// TIA Portal project "firstPro" (V15)

(* hardware
DEVICE "S71500/ET200MP station_1"  S7-1500 station
   slot 0: "导轨_0"  Rack  6ES7 590-1***0-0AA0
   slot 1: "PLC_1"  CPU 1516-3 PN/DP  6ES7 516-3AN01-0AB0  V2.5
      slot 3: "CPU 显示_1"  6ES7591-1BA00-0AA0
*)

// ===== PLC "PLC_1"  CPU 1516-3 PN/DP =====

VAR_GLOBAL   // PLC tag table "默认变量表"
   "targetdownFlag" AT %M1.0 : Bool;
   "targetupFlag" AT %M1.1 : Bool;
   "targetstopFlag" AT %M1.2 : Bool;
   "Tag_1" AT %T1 : Timer;
END_VAR

VAR_GLOBAL   // PLC tag table "变量表_1"
   "1 层上行呼梯按钮储存值" AT %I0.0 : Bool;
   "2 层上行呼梯按钮储存值" AT %I0.1 : Bool;
   "3 层上行呼梯按钮储存值" AT %I0.2 : Bool;
   "4 层上行呼梯按钮储存值" AT %I0.3 : Bool;
   "5 层上行呼梯按钮储存值" AT %I0.4 : Bool;
   "2 层下行呼梯按钮储存值" AT %I0.5 : Bool;
   "3 层下行呼梯按钮储存值" AT %I0.6 : Bool;
   "4 层下行呼梯按钮储存值" AT %I0.7 : Bool;
   "5 层下行呼梯按钮储存值" AT %I1.0 : Bool;
   "6 层下行呼梯按钮储存值" AT %I1.1 : Bool;
   "1 号梯轿内选层按钮 1储存值" AT %I1.2 : Bool;
   "1 号梯轿内选层按钮 2储存值" AT %I1.3 : Bool;
   "1 号梯轿内选层按钮 3储存值" AT %I1.4 : Bool;
   "1 号梯轿内选层按钮 4储存值" AT %I1.5 : Bool;
   "1 号梯轿内选层按钮 5储存值" AT %I1.6 : Bool;
   "1 号梯轿内选层按钮 6储存值" AT %I1.7 : Bool;
   "1层是否登记" AT %I2.0 : Bool;
   "2层是否登记" AT %I2.1 : Bool;
   "3层是否登记" AT %I2.2 : Bool;
   "4层是否登记" AT %I2.3 : Bool;
   "5层是否登记" AT %I2.4 : Bool;
   "6层是否登记" AT %I2.5 : Bool;
   "开门按钮储存值" AT %I2.6 : Bool;
   "关门按钮储存值" AT %I2.7 : Bool;
   "上平层信号储存值1" AT %I3.0 : Bool;
   "下平层信号储存值1" AT %I3.1 : Bool;
   "上平层信号储存值2" AT %I3.2 : Bool;
   "下平层信号储存值2" AT %I3.3 : Bool;
END_VAR

DATA_BLOCK "input"   // DB1
{ S7_Optimized_Access := 'FALSE' }
VERSION : 0.1
   VAR
      "1 层上行呼梯按钮" : Bool;
      "2 层上行呼梯按钮" : Bool;
      "3 层上行呼梯按钮" : Bool;
      "4 层上行呼梯按钮" : Bool;
      "5 层上行呼梯按钮" : Bool;
      "2 层下行呼梯按钮" : Bool;
      "3 层下行呼梯按钮" : Bool;
      "4 层下行呼梯按钮" : Bool;
      "5 层下行呼梯按钮" : Bool;
      "6 层下行呼梯按钮" : Bool;
      "1 号梯轿内选层按钮 1" : Bool;
      "1 号梯轿内选层按钮 2" : Bool;
      "1 号梯轿内选层按钮 3" : Bool;
      "1 号梯轿内选层按钮 4" : Bool;
      "1 号梯轿内选层按钮 5" : Bool;
      "1 号梯轿内选层按钮 6" : Bool;
      "1 号梯轿内开门按钮" : Bool;
      "1 号梯轿内关门按钮" : Bool;
      "1 号梯光幕信号" : Bool;
      "1 号梯检修信号" : Bool;
      "1 号梯轿厢门锁信号" : Bool;
      "1 号梯 1 楼层门锁信号" : Bool;
      "1 号梯 2 楼层门锁信号" : Bool;
      "1 号梯 3 楼层门锁信号" : Bool;
      "1 号梯 4 楼层门锁信号" : Bool;
      "1 号梯 5 楼层门锁信号" : Bool;
      "1 号梯 6 楼层门锁信号" : Bool;
      "1 号梯开门到位" : Bool;
      "1 号梯关门到位" : Bool;
      "1 号梯上平层信号" : Bool;
      "1 号梯下平层信号" : Bool;
      "1 号梯上端站第 1 限位" : Bool;
      "1 号梯上端站第 2 限位" : Bool;
      "1 号梯下端站第 1 限位" : Bool;
      "1 号梯下端站第 2 限位" : Bool;
      自动运行信号 : Bool;
      "1 号梯当前载重量" : Word := 0;
   END_VAR
BEGIN
END_DATA_BLOCK

DATA_BLOCK "output"   // DB2
{ S7_Optimized_Access := 'FALSE' }
VERSION : 0.1
   VAR
      "1 层上行呼梯按钮指示灯" : Bool;
      "2 层上行呼梯按钮指示灯" : Bool;
      "3 层上行呼梯按钮指示灯" : Bool;
      "4 层上行呼梯按钮指示灯" : Bool;
      "5 层上行呼梯按钮指示灯" : Bool;
      "2 层下行呼梯按钮指示灯" : Bool;
      "3 层下行呼梯按钮指示灯" : Bool;
      "4 层下行呼梯按钮指示灯" : Bool;
      "5 层下行呼梯按钮指示灯" : Bool;
      "6 层下行呼梯按钮指示灯" : Bool;
      "1 号梯 1 层按钮指示灯" : Bool;
      "1 号梯 2 层按钮指示灯" : Bool;
      "1 号梯 3 层按钮指示灯" : Bool;
      "1 号梯 4 层按钮指示灯" : Bool;
      "1 号梯 5 层按钮指示灯" : Bool;
      "1 号梯 6 层按钮指示灯" : Bool;
      "1 号梯 LEDa" : Bool;
      "1 号梯 LEDb" : Bool;
      "1 号梯 LEDc" : Bool;
      "1 号梯 LEDd" : Bool;
      "1 号梯 LEDe" : Bool;
      "1 号梯 LEDf" : Bool;
      "1 号梯 LEDg" : Bool;
      "1 号梯上行指示" : Bool;
      "1 号梯下行指示" : Bool;
      "1 号梯故障指示" : Bool;
      "1 号梯照明指示" : Bool;
      "1 号梯风扇指示" : Bool;
      "1 号梯满载指示" : Bool;
      "1 号梯电机启动信号" : Bool;
      "1 号梯上行接触器" : Bool;
      "1 号梯下行接触器" : Bool;
      "1 号梯高速接触器" : Bool;
      "1 号梯低速接触器" : Bool;
      "1 号梯开门继电器" : Bool;
      "1 号梯关门继电器" : Bool;
      "1 号梯 1 级减速制动" : Bool;
      "1 号梯 2 级减速制动" : Bool;
      "1 号梯 3 级减速制动" : Bool;
      准备就绪信号 : Bool;
   END_VAR
BEGIN
END_DATA_BLOCK

DATA_BLOCK "StateFlag"   // DB3
{ S7_Optimized_Access := 'TRUE' }
VERSION : 0.1
   VAR
      upwardFlag : Bool;
      breakingFlag : Bool;
      downwardFlag : Bool;
      startupState : UInt;
      startupflag : Bool;
      upwardState : Bool;
      downwardState : Bool;
      折返指示 : UInt;
      "1层是否登记" : Bool;
      "2层是否登记" : Bool;
      "3层是否登记" : Bool;
      "4层是否登记" : Bool;
      "5层是否登记" : Bool;
      "6层是否登记" : Bool;
      楼层是否登记 : Byte;
      重置上下行指示 : Bool := true;
      检修状态 : UInt;
   END_VAR
BEGIN
END_DATA_BLOCK

DATA_BLOCK "liftInfo"   // DB4
{ S7_Optimized_Access := 'TRUE' }
VERSION : 0.1
   VAR
      floor : Byte := 16#0;
      tartget : Byte := 16#0;
      楼层登记 : Byte;
      等待上行到达目标 : Bool;
      等待下行到达目标 : Bool;
      上行登记 : Byte;
      下行登记 : Byte;
      停层信号 : Bool;
      开门按钮储存位 : Bool;
      关门按钮储存位 : Bool;
      开门锁上下行 : Bool;
      空闲状态 : Bool := true;
      门锁信号 : Bool;
      复位空闲状态 : Bool;
      梯内按钮输入 : Byte;
      上行按钮输入 : Byte;
      下行按钮输入 : Byte;
      上下行指示 : Byte;
      上行登记掩码 : Byte := 16#3F;
      下行登记掩码 : Byte;
      检修信号 : Bool;
   END_VAR
BEGIN
END_DATA_BLOCK

DATA_BLOCK "指示灯_DB"   // DB5
{ S7_Optimized_Access := 'TRUE' }
VERSION : 0.1
// stored: InstanceOfName 指示灯
"指示灯"
BEGIN
END_DATA_BLOCK

DATA_BLOCK "constant"   // DB6
{ S7_Optimized_Access := 'TRUE' }
VERSION : 0.1
   VAR
      "1楼登记" : Byte := 16#1;
      "2楼登记" : Byte := 16#2;
      "3楼登记" : Byte := 16#4;
      "4楼登记" : Byte := 16#8;
      "5楼登记" : Byte := 16#10;
      "6楼登记" : Byte := 16#20;
      上行 : Bool := true;
      下行 : Bool;
      梯内按钮输入掩码 : Byte := 16#3F;
      上行按钮输入掩码 : Byte := 16#1F;
      下行按钮输入掩码 : Byte := 16#3F;
      楼层掩码 : Byte := 16#3F;
      上下行指示掩码 : Byte := 16#3;
      梯内按钮输入 : UInt;
      上行按钮输入 : UInt := 1;
      下行按钮输入 : UInt := 2;
      当前楼层 : UInt := 3;
      目标楼层 : UInt := 4;
      上下行指示 : UInt := 5;
      "1楼" : Byte := 16#1;
      "2楼" : Byte := 16#2;
      "3楼" : Byte := 16#4;
      "4楼" : Byte := 16#8;
      "5楼" : Byte := 16#10;
      "6楼" : Byte := 16#20;
   END_VAR
BEGIN
END_DATA_BLOCK

DATA_BLOCK "错误检测_DB"   // DB7
{ S7_Optimized_Access := 'TRUE' }
VERSION : 0.1
// stored: InstanceOfName 错误检测
"错误检测"
BEGIN
END_DATA_BLOCK

DATA_BLOCK "电梯上下行控制_DB_1"   // DB8
{ S7_Optimized_Access := 'TRUE' }
VERSION : 0.1
// stored: InstanceOfName 电梯上下行控制
"电梯上下行控制"
BEGIN
END_DATA_BLOCK

DATA_BLOCK "开关门_DB"   // DB10
{ S7_Optimized_Access := 'TRUE' }
VERSION : 0.1
// stored: InstanceOfName 开关门
"开关门"
BEGIN
END_DATA_BLOCK

DATA_BLOCK "外部信号处理储存值"   // DB16
{ S7_Optimized_Access := 'TRUE' }
VERSION : 0.1
   VAR
      梯内按钮遍历层 : Byte := 16#1;
      上行按钮遍历层 : Byte := 16#1;
      下行按钮遍历层 : Byte := 16#2;
   END_VAR
BEGIN
END_DATA_BLOCK

// folder: System blocks/Program resources

DATA_BLOCK "IEC_Timer_0_DB"   // DB9
{ S7_Optimized_Access := 'TRUE' }
AUTHOR : Simatic
FAMILY : IEC
NAME : IEC_TMR
VERSION : 1.0
// stored: InstanceOfName IEC_TIMER
"IEC_TIMER"
BEGIN
END_DATA_BLOCK

DATA_BLOCK "IEC_Timer_0_DB_2"   // DB11
{ S7_Optimized_Access := 'TRUE' }
AUTHOR : Simatic
FAMILY : IEC
NAME : IEC_TMR
VERSION : 1.0
// stored: InstanceOfName IEC_TIMER
"IEC_TIMER"
BEGIN
END_DATA_BLOCK

DATA_BLOCK "IEC_Timer_0_DB_3"   // DB12
{ S7_Optimized_Access := 'TRUE' }
AUTHOR : Simatic
FAMILY : IEC
NAME : IEC_TMR
VERSION : 1.0
// stored: InstanceOfName IEC_TIMER
"IEC_TIMER"
BEGIN
END_DATA_BLOCK

DATA_BLOCK "IEC_Timer_0_DB_4"   // DB13
{ S7_Optimized_Access := 'TRUE' }
AUTHOR : Simatic
FAMILY : IEC
NAME : IEC_TMR
VERSION : 1.0
// stored: InstanceOfName IEC_TIMER
"IEC_TIMER"
BEGIN
END_DATA_BLOCK

DATA_BLOCK "IEC_Timer_0_DB_5"   // DB14
{ S7_Optimized_Access := 'TRUE' }
AUTHOR : Simatic
FAMILY : IEC
NAME : IEC_TMR
VERSION : 1.0
// stored: InstanceOfName IEC_TIMER
"IEC_TIMER"
BEGIN
END_DATA_BLOCK

DATA_BLOCK "IEC_Timer_0_DB_1"   // DB15
{ S7_Optimized_Access := 'TRUE' }
AUTHOR : Simatic
FAMILY : IEC
NAME : IEC_TMR
VERSION : 1.0
// stored: InstanceOfName IEC_TIMER
"IEC_TIMER"
BEGIN
END_DATA_BLOCK

// folder: (top level)

FUNCTION_BLOCK "指示灯"   // FB1, LAD
{ S7_Optimized_Access := 'TRUE' }
VERSION : 0.1
   VAR_TEMP
      tmp1 : Bool;
   END_VAR
   VAR_TEMP   // added for the SCL form of the ladder/FBD networks
      _w1 : Bool;
      _w2 : Bool;
   END_VAR
BEGIN

REGION Network 1: 1层上行按钮
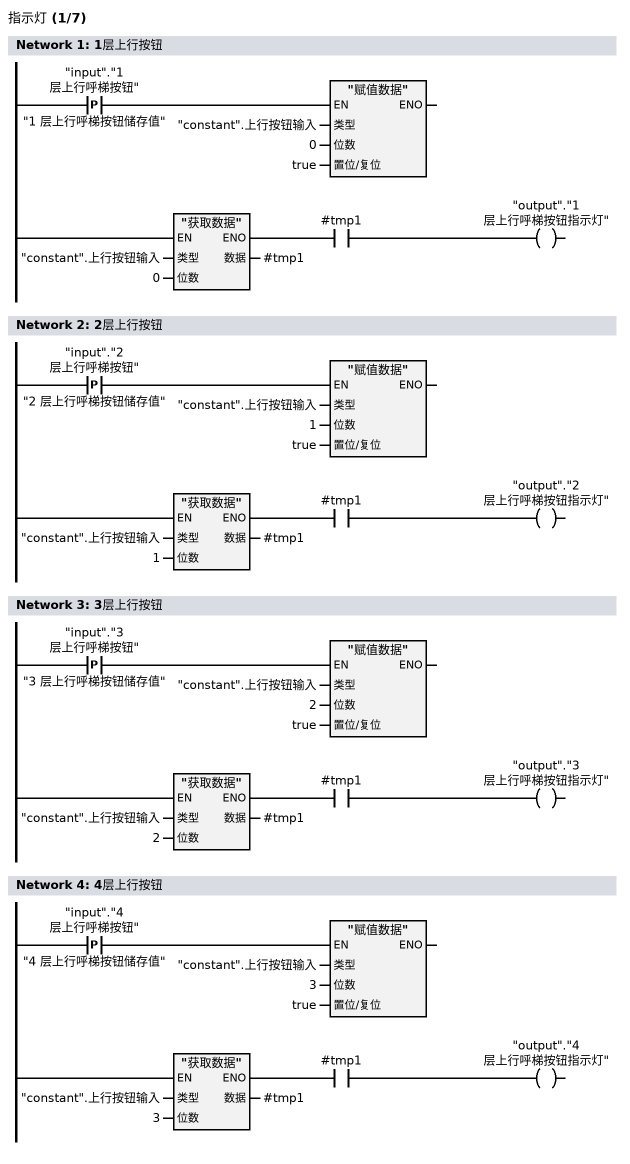
   RUNG wire#powerrail
      P_Contact(operand := "input"."1 层上行呼梯按钮", bit := "1 层上行呼梯按钮储存值")
      "赋值数据"(类型 := "constant".上行按钮输入, 位数 := 0, "置位/复位" := true)
   END_RUNG
   RUNG wire#powerrail
      "获取数据"(类型 := "constant".上行按钮输入, 位数 := 0, 数据 => #tmp1)
      Contact( #tmp1 )
      Coil( "output"."1 层上行呼梯按钮指示灯" )
   END_RUNG
   // the same network as SCL:
   #_w1 := "input"."1 层上行呼梯按钮" AND NOT "1 层上行呼梯按钮储存值";   // rising edge of "input"."1 层上行呼梯按钮"
   "1 层上行呼梯按钮储存值" := "input"."1 层上行呼梯按钮";
   IF #_w1 THEN "赋值数据"(类型 := "constant".上行按钮输入, 位数 := 0, "置位/复位" := true); END_IF;
   "获取数据"(类型 := "constant".上行按钮输入, 位数 := 0, 数据 => #tmp1, ENO => #_w2);
   "output"."1 层上行呼梯按钮指示灯" := #_w2 AND #tmp1;
END_REGION

REGION Network 2: 2层上行按钮
   RUNG wire#powerrail
      P_Contact(operand := "input"."2 层上行呼梯按钮", bit := "2 层上行呼梯按钮储存值")
      "赋值数据"(类型 := "constant".上行按钮输入, 位数 := 1, "置位/复位" := true)
   END_RUNG
   RUNG wire#powerrail
      "获取数据"(类型 := "constant".上行按钮输入, 位数 := 1, 数据 => #tmp1)
      Contact( #tmp1 )
      Coil( "output"."2 层上行呼梯按钮指示灯" )
   END_RUNG
   // the same network as SCL:
   #_w1 := "input"."2 层上行呼梯按钮" AND NOT "2 层上行呼梯按钮储存值";   // rising edge of "input"."2 层上行呼梯按钮"
   "2 层上行呼梯按钮储存值" := "input"."2 层上行呼梯按钮";
   IF #_w1 THEN "赋值数据"(类型 := "constant".上行按钮输入, 位数 := 1, "置位/复位" := true); END_IF;
   "获取数据"(类型 := "constant".上行按钮输入, 位数 := 1, 数据 => #tmp1, ENO => #_w2);
   "output"."2 层上行呼梯按钮指示灯" := #_w2 AND #tmp1;
END_REGION

REGION Network 3: 3层上行按钮
   RUNG wire#powerrail
      P_Contact(operand := "input"."3 层上行呼梯按钮", bit := "3 层上行呼梯按钮储存值")
      "赋值数据"(类型 := "constant".上行按钮输入, 位数 := 2, "置位/复位" := true)
   END_RUNG
   RUNG wire#powerrail
      "获取数据"(类型 := "constant".上行按钮输入, 位数 := 2, 数据 => #tmp1)
      Contact( #tmp1 )
      Coil( "output"."3 层上行呼梯按钮指示灯" )
   END_RUNG
   // the same network as SCL:
   #_w1 := "input"."3 层上行呼梯按钮" AND NOT "3 层上行呼梯按钮储存值";   // rising edge of "input"."3 层上行呼梯按钮"
   "3 层上行呼梯按钮储存值" := "input"."3 层上行呼梯按钮";
   IF #_w1 THEN "赋值数据"(类型 := "constant".上行按钮输入, 位数 := 2, "置位/复位" := true); END_IF;
   "获取数据"(类型 := "constant".上行按钮输入, 位数 := 2, 数据 => #tmp1, ENO => #_w2);
   "output"."3 层上行呼梯按钮指示灯" := #_w2 AND #tmp1;
END_REGION

REGION Network 4: 4层上行按钮
   RUNG wire#powerrail
      P_Contact(operand := "input"."4 层上行呼梯按钮", bit := "4 层上行呼梯按钮储存值")
      "赋值数据"(类型 := "constant".上行按钮输入, 位数 := 3, "置位/复位" := true)
   END_RUNG
   RUNG wire#powerrail
      "获取数据"(类型 := "constant".上行按钮输入, 位数 := 3, 数据 => #tmp1)
      Contact( #tmp1 )
      Coil( "output"."4 层上行呼梯按钮指示灯" )
   END_RUNG
   // the same network as SCL:
   #_w1 := "input"."4 层上行呼梯按钮" AND NOT "4 层上行呼梯按钮储存值";   // rising edge of "input"."4 层上行呼梯按钮"
   "4 层上行呼梯按钮储存值" := "input"."4 层上行呼梯按钮";
   IF #_w1 THEN "赋值数据"(类型 := "constant".上行按钮输入, 位数 := 3, "置位/复位" := true); END_IF;
   "获取数据"(类型 := "constant".上行按钮输入, 位数 := 3, 数据 => #tmp1, ENO => #_w2);
   "output"."4 层上行呼梯按钮指示灯" := #_w2 AND #tmp1;
END_REGION

REGION Network 5: 5层上行按钮
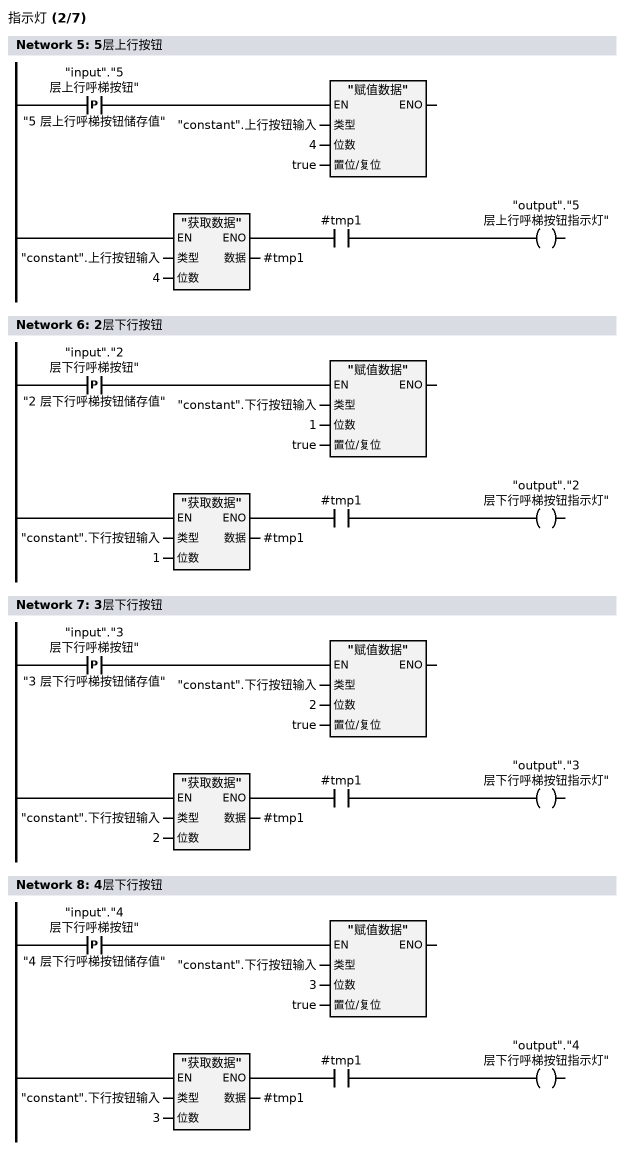
   RUNG wire#powerrail
      P_Contact(operand := "input"."5 层上行呼梯按钮", bit := "5 层上行呼梯按钮储存值")
      "赋值数据"(类型 := "constant".上行按钮输入, 位数 := 4, "置位/复位" := true)
   END_RUNG
   RUNG wire#powerrail
      "获取数据"(类型 := "constant".上行按钮输入, 位数 := 4, 数据 => #tmp1)
      Contact( #tmp1 )
      Coil( "output"."5 层上行呼梯按钮指示灯" )
   END_RUNG
   // the same network as SCL:
   #_w1 := "input"."5 层上行呼梯按钮" AND NOT "5 层上行呼梯按钮储存值";   // rising edge of "input"."5 层上行呼梯按钮"
   "5 层上行呼梯按钮储存值" := "input"."5 层上行呼梯按钮";
   IF #_w1 THEN "赋值数据"(类型 := "constant".上行按钮输入, 位数 := 4, "置位/复位" := true); END_IF;
   "获取数据"(类型 := "constant".上行按钮输入, 位数 := 4, 数据 => #tmp1, ENO => #_w2);
   "output"."5 层上行呼梯按钮指示灯" := #_w2 AND #tmp1;
END_REGION

REGION Network 6: 2层下行按钮
   RUNG wire#powerrail
      P_Contact(operand := "input"."2 层下行呼梯按钮", bit := "2 层下行呼梯按钮储存值")
      "赋值数据"(类型 := "constant".下行按钮输入, 位数 := 1, "置位/复位" := true)
   END_RUNG
   RUNG wire#powerrail
      "获取数据"(类型 := "constant".下行按钮输入, 位数 := 1, 数据 => #tmp1)
      Contact( #tmp1 )
      Coil( "output"."2 层下行呼梯按钮指示灯" )
   END_RUNG
   // the same network as SCL:
   #_w1 := "input"."2 层下行呼梯按钮" AND NOT "2 层下行呼梯按钮储存值";   // rising edge of "input"."2 层下行呼梯按钮"
   "2 层下行呼梯按钮储存值" := "input"."2 层下行呼梯按钮";
   IF #_w1 THEN "赋值数据"(类型 := "constant".下行按钮输入, 位数 := 1, "置位/复位" := true); END_IF;
   "获取数据"(类型 := "constant".下行按钮输入, 位数 := 1, 数据 => #tmp1, ENO => #_w2);
   "output"."2 层下行呼梯按钮指示灯" := #_w2 AND #tmp1;
END_REGION

REGION Network 7: 3层下行按钮
   RUNG wire#powerrail
      P_Contact(operand := "input"."3 层下行呼梯按钮", bit := "3 层下行呼梯按钮储存值")
      "赋值数据"(类型 := "constant".下行按钮输入, 位数 := 2, "置位/复位" := true)
   END_RUNG
   RUNG wire#powerrail
      "获取数据"(类型 := "constant".下行按钮输入, 位数 := 2, 数据 => #tmp1)
      Contact( #tmp1 )
      Coil( "output"."3 层下行呼梯按钮指示灯" )
   END_RUNG
   // the same network as SCL:
   #_w1 := "input"."3 层下行呼梯按钮" AND NOT "3 层下行呼梯按钮储存值";   // rising edge of "input"."3 层下行呼梯按钮"
   "3 层下行呼梯按钮储存值" := "input"."3 层下行呼梯按钮";
   IF #_w1 THEN "赋值数据"(类型 := "constant".下行按钮输入, 位数 := 2, "置位/复位" := true); END_IF;
   "获取数据"(类型 := "constant".下行按钮输入, 位数 := 2, 数据 => #tmp1, ENO => #_w2);
   "output"."3 层下行呼梯按钮指示灯" := #_w2 AND #tmp1;
END_REGION

REGION Network 8: 4层下行按钮
   RUNG wire#powerrail
      P_Contact(operand := "input"."4 层下行呼梯按钮", bit := "4 层下行呼梯按钮储存值")
      "赋值数据"(类型 := "constant".下行按钮输入, 位数 := 3, "置位/复位" := true)
   END_RUNG
   RUNG wire#powerrail
      "获取数据"(类型 := "constant".下行按钮输入, 位数 := 3, 数据 => #tmp1)
      Contact( #tmp1 )
      Coil( "output"."4 层下行呼梯按钮指示灯" )
   END_RUNG
   // the same network as SCL:
   #_w1 := "input"."4 层下行呼梯按钮" AND NOT "4 层下行呼梯按钮储存值";   // rising edge of "input"."4 层下行呼梯按钮"
   "4 层下行呼梯按钮储存值" := "input"."4 层下行呼梯按钮";
   IF #_w1 THEN "赋值数据"(类型 := "constant".下行按钮输入, 位数 := 3, "置位/复位" := true); END_IF;
   "获取数据"(类型 := "constant".下行按钮输入, 位数 := 3, 数据 => #tmp1, ENO => #_w2);
   "output"."4 层下行呼梯按钮指示灯" := #_w2 AND #tmp1;
END_REGION

REGION Network 9: 5层下行按钮
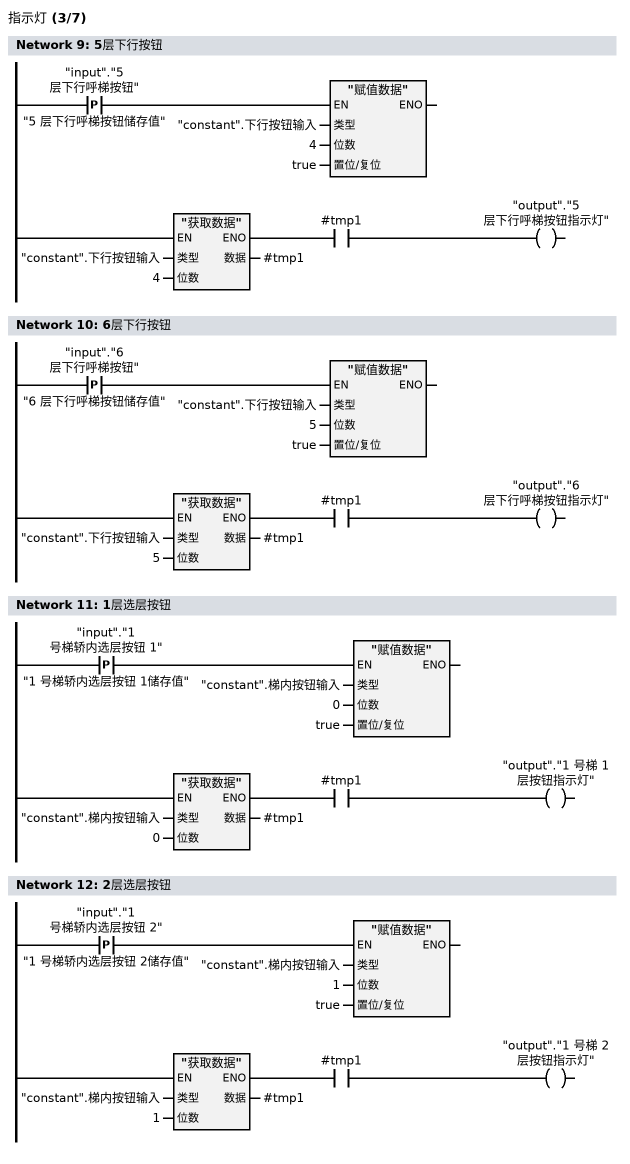
   RUNG wire#powerrail
      P_Contact(operand := "input"."5 层下行呼梯按钮", bit := "5 层下行呼梯按钮储存值")
      "赋值数据"(类型 := "constant".下行按钮输入, 位数 := 4, "置位/复位" := true)
   END_RUNG
   RUNG wire#powerrail
      "获取数据"(类型 := "constant".下行按钮输入, 位数 := 4, 数据 => #tmp1)
      Contact( #tmp1 )
      Coil( "output"."5 层下行呼梯按钮指示灯" )
   END_RUNG
   // the same network as SCL:
   #_w1 := "input"."5 层下行呼梯按钮" AND NOT "5 层下行呼梯按钮储存值";   // rising edge of "input"."5 层下行呼梯按钮"
   "5 层下行呼梯按钮储存值" := "input"."5 层下行呼梯按钮";
   IF #_w1 THEN "赋值数据"(类型 := "constant".下行按钮输入, 位数 := 4, "置位/复位" := true); END_IF;
   "获取数据"(类型 := "constant".下行按钮输入, 位数 := 4, 数据 => #tmp1, ENO => #_w2);
   "output"."5 层下行呼梯按钮指示灯" := #_w2 AND #tmp1;
END_REGION

REGION Network 10: 6层下行按钮
   RUNG wire#powerrail
      P_Contact(operand := "input"."6 层下行呼梯按钮", bit := "6 层下行呼梯按钮储存值")
      "赋值数据"(类型 := "constant".下行按钮输入, 位数 := 5, "置位/复位" := true)
   END_RUNG
   RUNG wire#powerrail
      "获取数据"(类型 := "constant".下行按钮输入, 位数 := 5, 数据 => #tmp1)
      Contact( #tmp1 )
      Coil( "output"."6 层下行呼梯按钮指示灯" )
   END_RUNG
   // the same network as SCL:
   #_w1 := "input"."6 层下行呼梯按钮" AND NOT "6 层下行呼梯按钮储存值";   // rising edge of "input"."6 层下行呼梯按钮"
   "6 层下行呼梯按钮储存值" := "input"."6 层下行呼梯按钮";
   IF #_w1 THEN "赋值数据"(类型 := "constant".下行按钮输入, 位数 := 5, "置位/复位" := true); END_IF;
   "获取数据"(类型 := "constant".下行按钮输入, 位数 := 5, 数据 => #tmp1, ENO => #_w2);
   "output"."6 层下行呼梯按钮指示灯" := #_w2 AND #tmp1;
END_REGION

REGION Network 11: 1层选层按钮
   RUNG wire#powerrail
      P_Contact(operand := "input"."1 号梯轿内选层按钮 1", bit := "1 号梯轿内选层按钮 1储存值")
      "赋值数据"(类型 := "constant".梯内按钮输入, 位数 := 0, "置位/复位" := true)
   END_RUNG
   RUNG wire#powerrail
      "获取数据"(类型 := "constant".梯内按钮输入, 位数 := 0, 数据 => #tmp1)
      Contact( #tmp1 )
      Coil( "output"."1 号梯 1 层按钮指示灯" )
   END_RUNG
   // the same network as SCL:
   #_w1 := "input"."1 号梯轿内选层按钮 1" AND NOT "1 号梯轿内选层按钮 1储存值";   // rising edge of "input"."1 号梯轿内选层按钮 1"
   "1 号梯轿内选层按钮 1储存值" := "input"."1 号梯轿内选层按钮 1";
   IF #_w1 THEN "赋值数据"(类型 := "constant".梯内按钮输入, 位数 := 0, "置位/复位" := true); END_IF;
   "获取数据"(类型 := "constant".梯内按钮输入, 位数 := 0, 数据 => #tmp1, ENO => #_w2);
   "output"."1 号梯 1 层按钮指示灯" := #_w2 AND #tmp1;
END_REGION

REGION Network 12: 2层选层按钮
   RUNG wire#powerrail
      P_Contact(operand := "input"."1 号梯轿内选层按钮 2", bit := "1 号梯轿内选层按钮 2储存值")
      "赋值数据"(类型 := "constant".梯内按钮输入, 位数 := 1, "置位/复位" := true)
   END_RUNG
   RUNG wire#powerrail
      "获取数据"(类型 := "constant".梯内按钮输入, 位数 := 1, 数据 => #tmp1)
      Contact( #tmp1 )
      Coil( "output"."1 号梯 2 层按钮指示灯" )
   END_RUNG
   // the same network as SCL:
   #_w1 := "input"."1 号梯轿内选层按钮 2" AND NOT "1 号梯轿内选层按钮 2储存值";   // rising edge of "input"."1 号梯轿内选层按钮 2"
   "1 号梯轿内选层按钮 2储存值" := "input"."1 号梯轿内选层按钮 2";
   IF #_w1 THEN "赋值数据"(类型 := "constant".梯内按钮输入, 位数 := 1, "置位/复位" := true); END_IF;
   "获取数据"(类型 := "constant".梯内按钮输入, 位数 := 1, 数据 => #tmp1, ENO => #_w2);
   "output"."1 号梯 2 层按钮指示灯" := #_w2 AND #tmp1;
END_REGION

REGION Network 13: 3层选层按钮
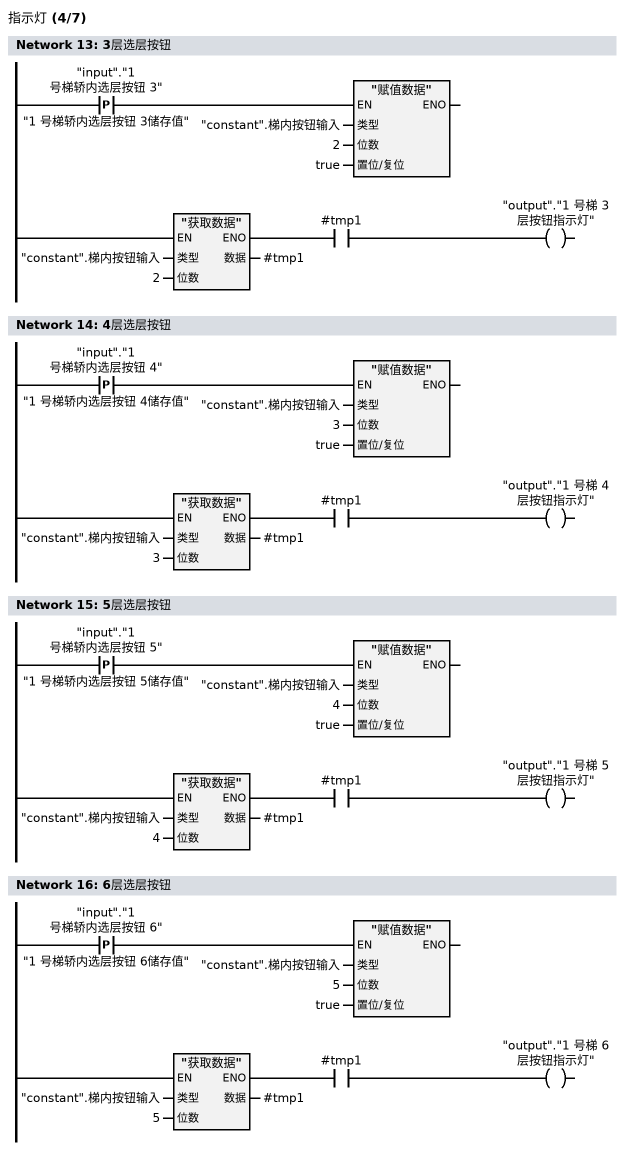
   RUNG wire#powerrail
      P_Contact(operand := "input"."1 号梯轿内选层按钮 3", bit := "1 号梯轿内选层按钮 3储存值")
      "赋值数据"(类型 := "constant".梯内按钮输入, 位数 := 2, "置位/复位" := true)
   END_RUNG
   RUNG wire#powerrail
      "获取数据"(类型 := "constant".梯内按钮输入, 位数 := 2, 数据 => #tmp1)
      Contact( #tmp1 )
      Coil( "output"."1 号梯 3 层按钮指示灯" )
   END_RUNG
   // the same network as SCL:
   #_w1 := "input"."1 号梯轿内选层按钮 3" AND NOT "1 号梯轿内选层按钮 3储存值";   // rising edge of "input"."1 号梯轿内选层按钮 3"
   "1 号梯轿内选层按钮 3储存值" := "input"."1 号梯轿内选层按钮 3";
   IF #_w1 THEN "赋值数据"(类型 := "constant".梯内按钮输入, 位数 := 2, "置位/复位" := true); END_IF;
   "获取数据"(类型 := "constant".梯内按钮输入, 位数 := 2, 数据 => #tmp1, ENO => #_w2);
   "output"."1 号梯 3 层按钮指示灯" := #_w2 AND #tmp1;
END_REGION

REGION Network 14: 4层选层按钮
   RUNG wire#powerrail
      P_Contact(operand := "input"."1 号梯轿内选层按钮 4", bit := "1 号梯轿内选层按钮 4储存值")
      "赋值数据"(类型 := "constant".梯内按钮输入, 位数 := 3, "置位/复位" := true)
   END_RUNG
   RUNG wire#powerrail
      "获取数据"(类型 := "constant".梯内按钮输入, 位数 := 3, 数据 => #tmp1)
      Contact( #tmp1 )
      Coil( "output"."1 号梯 4 层按钮指示灯" )
   END_RUNG
   // the same network as SCL:
   #_w1 := "input"."1 号梯轿内选层按钮 4" AND NOT "1 号梯轿内选层按钮 4储存值";   // rising edge of "input"."1 号梯轿内选层按钮 4"
   "1 号梯轿内选层按钮 4储存值" := "input"."1 号梯轿内选层按钮 4";
   IF #_w1 THEN "赋值数据"(类型 := "constant".梯内按钮输入, 位数 := 3, "置位/复位" := true); END_IF;
   "获取数据"(类型 := "constant".梯内按钮输入, 位数 := 3, 数据 => #tmp1, ENO => #_w2);
   "output"."1 号梯 4 层按钮指示灯" := #_w2 AND #tmp1;
END_REGION

REGION Network 15: 5层选层按钮
   RUNG wire#powerrail
      P_Contact(operand := "input"."1 号梯轿内选层按钮 5", bit := "1 号梯轿内选层按钮 5储存值")
      "赋值数据"(类型 := "constant".梯内按钮输入, 位数 := 4, "置位/复位" := true)
   END_RUNG
   RUNG wire#powerrail
      "获取数据"(类型 := "constant".梯内按钮输入, 位数 := 4, 数据 => #tmp1)
      Contact( #tmp1 )
      Coil( "output"."1 号梯 5 层按钮指示灯" )
   END_RUNG
   // the same network as SCL:
   #_w1 := "input"."1 号梯轿内选层按钮 5" AND NOT "1 号梯轿内选层按钮 5储存值";   // rising edge of "input"."1 号梯轿内选层按钮 5"
   "1 号梯轿内选层按钮 5储存值" := "input"."1 号梯轿内选层按钮 5";
   IF #_w1 THEN "赋值数据"(类型 := "constant".梯内按钮输入, 位数 := 4, "置位/复位" := true); END_IF;
   "获取数据"(类型 := "constant".梯内按钮输入, 位数 := 4, 数据 => #tmp1, ENO => #_w2);
   "output"."1 号梯 5 层按钮指示灯" := #_w2 AND #tmp1;
END_REGION

REGION Network 16: 6层选层按钮
   RUNG wire#powerrail
      P_Contact(operand := "input"."1 号梯轿内选层按钮 6", bit := "1 号梯轿内选层按钮 6储存值")
      "赋值数据"(类型 := "constant".梯内按钮输入, 位数 := 5, "置位/复位" := true)
   END_RUNG
   RUNG wire#powerrail
      "获取数据"(类型 := "constant".梯内按钮输入, 位数 := 5, 数据 => #tmp1)
      Contact( #tmp1 )
      Coil( "output"."1 号梯 6 层按钮指示灯" )
   END_RUNG
   // the same network as SCL:
   #_w1 := "input"."1 号梯轿内选层按钮 6" AND NOT "1 号梯轿内选层按钮 6储存值";   // rising edge of "input"."1 号梯轿内选层按钮 6"
   "1 号梯轿内选层按钮 6储存值" := "input"."1 号梯轿内选层按钮 6";
   IF #_w1 THEN "赋值数据"(类型 := "constant".梯内按钮输入, 位数 := 5, "置位/复位" := true); END_IF;
   "获取数据"(类型 := "constant".梯内按钮输入, 位数 := 5, 数据 => #tmp1, ENO => #_w2);
   "output"."1 号梯 6 层按钮指示灯" := #_w2 AND #tmp1;
END_REGION

REGION Network 17: One
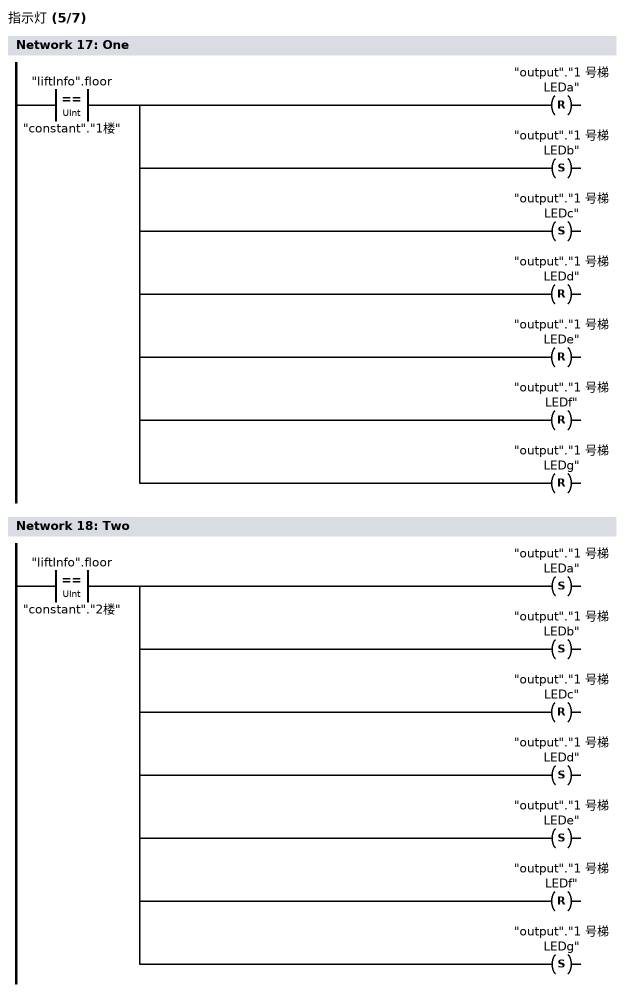
   RUNG wire#powerrail
      { S7_Templates := "SrcType := UInt" } EQ_Contact(in1 := "liftInfo".floor, in2 := "constant"."1楼")
      wire#w1
      R_Coil( "output"."1 号梯 LEDa" )
   END_RUNG
   RUNG wire#w1
      S_Coil( "output"."1 号梯 LEDb" )
   END_RUNG
   RUNG wire#w1
      S_Coil( "output"."1 号梯 LEDc" )
   END_RUNG
   RUNG wire#w1
      R_Coil( "output"."1 号梯 LEDd" )
   END_RUNG
   RUNG wire#w1
      R_Coil( "output"."1 号梯 LEDe" )
   END_RUNG
   RUNG wire#w1
      R_Coil( "output"."1 号梯 LEDf" )
   END_RUNG
   RUNG wire#w1
      R_Coil( "output"."1 号梯 LEDg" )
   END_RUNG
   // the same network as SCL:
   IF "liftInfo".floor = "constant"."1楼" THEN
       "output"."1 号梯 LEDa" := FALSE;
       "output"."1 号梯 LEDb" := TRUE;
       "output"."1 号梯 LEDc" := TRUE;
       "output"."1 号梯 LEDd" := FALSE;
       "output"."1 号梯 LEDe" := FALSE;
       "output"."1 号梯 LEDf" := FALSE;
       "output"."1 号梯 LEDg" := FALSE;
   END_IF;
END_REGION

REGION Network 18: Two
   RUNG wire#powerrail
      { S7_Templates := "SrcType := UInt" } EQ_Contact(in1 := "liftInfo".floor, in2 := "constant"."2楼")
      wire#w1
      S_Coil( "output"."1 号梯 LEDa" )
   END_RUNG
   RUNG wire#w1
      S_Coil( "output"."1 号梯 LEDb" )
   END_RUNG
   RUNG wire#w1
      R_Coil( "output"."1 号梯 LEDc" )
   END_RUNG
   RUNG wire#w1
      S_Coil( "output"."1 号梯 LEDd" )
   END_RUNG
   RUNG wire#w1
      S_Coil( "output"."1 号梯 LEDe" )
   END_RUNG
   RUNG wire#w1
      R_Coil( "output"."1 号梯 LEDf" )
   END_RUNG
   RUNG wire#w1
      S_Coil( "output"."1 号梯 LEDg" )
   END_RUNG
   // the same network as SCL:
   IF "liftInfo".floor = "constant"."2楼" THEN
       "output"."1 号梯 LEDa" := TRUE;
       "output"."1 号梯 LEDb" := TRUE;
       "output"."1 号梯 LEDc" := FALSE;
       "output"."1 号梯 LEDd" := TRUE;
       "output"."1 号梯 LEDe" := TRUE;
       "output"."1 号梯 LEDf" := FALSE;
       "output"."1 号梯 LEDg" := TRUE;
   END_IF;
END_REGION

REGION Network 19: Three
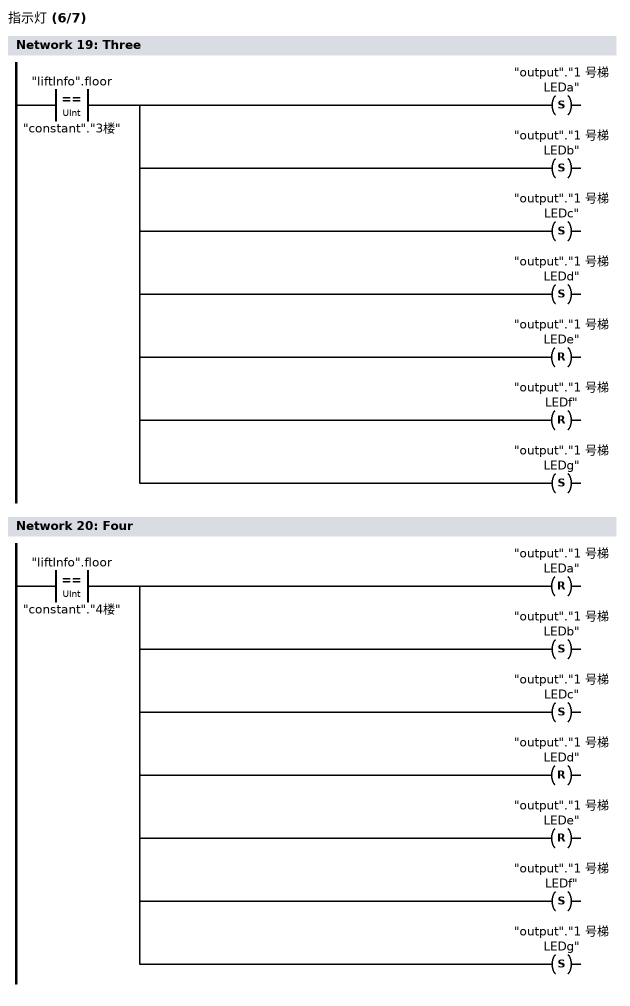
   RUNG wire#powerrail
      { S7_Templates := "SrcType := UInt" } EQ_Contact(in1 := "liftInfo".floor, in2 := "constant"."3楼")
      wire#w1
      S_Coil( "output"."1 号梯 LEDa" )
   END_RUNG
   RUNG wire#w1
      S_Coil( "output"."1 号梯 LEDb" )
   END_RUNG
   RUNG wire#w1
      S_Coil( "output"."1 号梯 LEDc" )
   END_RUNG
   RUNG wire#w1
      S_Coil( "output"."1 号梯 LEDd" )
   END_RUNG
   RUNG wire#w1
      R_Coil( "output"."1 号梯 LEDe" )
   END_RUNG
   RUNG wire#w1
      R_Coil( "output"."1 号梯 LEDf" )
   END_RUNG
   RUNG wire#w1
      S_Coil( "output"."1 号梯 LEDg" )
   END_RUNG
   // the same network as SCL:
   IF "liftInfo".floor = "constant"."3楼" THEN
       "output"."1 号梯 LEDa" := TRUE;
       "output"."1 号梯 LEDb" := TRUE;
       "output"."1 号梯 LEDc" := TRUE;
       "output"."1 号梯 LEDd" := TRUE;
       "output"."1 号梯 LEDe" := FALSE;
       "output"."1 号梯 LEDf" := FALSE;
       "output"."1 号梯 LEDg" := TRUE;
   END_IF;
END_REGION

REGION Network 20: Four
   RUNG wire#powerrail
      { S7_Templates := "SrcType := UInt" } EQ_Contact(in1 := "liftInfo".floor, in2 := "constant"."4楼")
      wire#w1
      R_Coil( "output"."1 号梯 LEDa" )
   END_RUNG
   RUNG wire#w1
      S_Coil( "output"."1 号梯 LEDb" )
   END_RUNG
   RUNG wire#w1
      S_Coil( "output"."1 号梯 LEDc" )
   END_RUNG
   RUNG wire#w1
      R_Coil( "output"."1 号梯 LEDd" )
   END_RUNG
   RUNG wire#w1
      R_Coil( "output"."1 号梯 LEDe" )
   END_RUNG
   RUNG wire#w1
      S_Coil( "output"."1 号梯 LEDf" )
   END_RUNG
   RUNG wire#w1
      S_Coil( "output"."1 号梯 LEDg" )
   END_RUNG
   // the same network as SCL:
   IF "liftInfo".floor = "constant"."4楼" THEN
       "output"."1 号梯 LEDa" := FALSE;
       "output"."1 号梯 LEDb" := TRUE;
       "output"."1 号梯 LEDc" := TRUE;
       "output"."1 号梯 LEDd" := FALSE;
       "output"."1 号梯 LEDe" := FALSE;
       "output"."1 号梯 LEDf" := TRUE;
       "output"."1 号梯 LEDg" := TRUE;
   END_IF;
END_REGION

REGION Network 21: Five
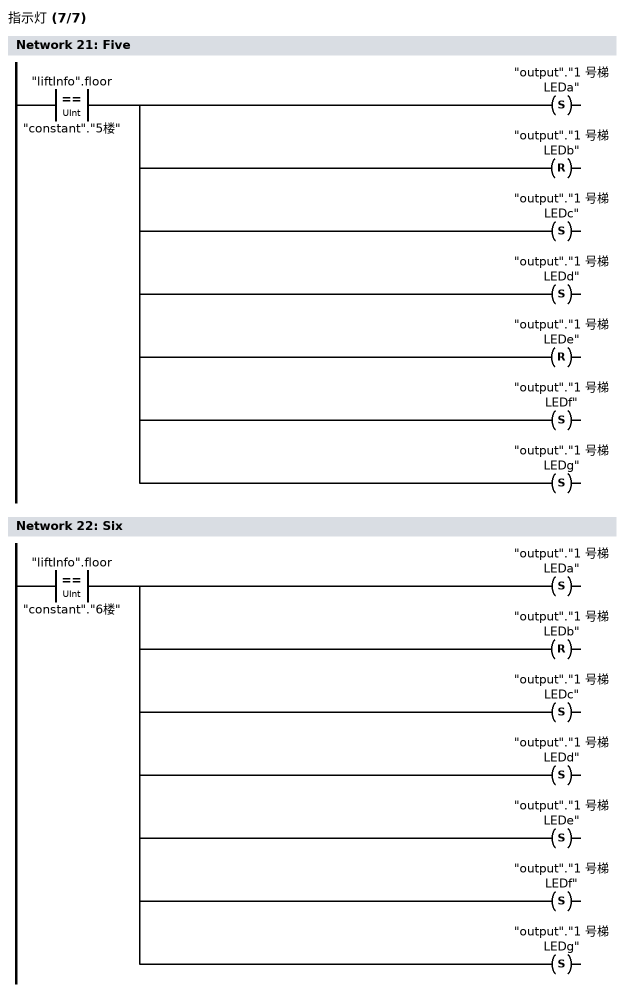
   RUNG wire#powerrail
      { S7_Templates := "SrcType := UInt" } EQ_Contact(in1 := "liftInfo".floor, in2 := "constant"."5楼")
      wire#w1
      S_Coil( "output"."1 号梯 LEDa" )
   END_RUNG
   RUNG wire#w1
      R_Coil( "output"."1 号梯 LEDb" )
   END_RUNG
   RUNG wire#w1
      S_Coil( "output"."1 号梯 LEDc" )
   END_RUNG
   RUNG wire#w1
      S_Coil( "output"."1 号梯 LEDd" )
   END_RUNG
   RUNG wire#w1
      R_Coil( "output"."1 号梯 LEDe" )
   END_RUNG
   RUNG wire#w1
      S_Coil( "output"."1 号梯 LEDf" )
   END_RUNG
   RUNG wire#w1
      S_Coil( "output"."1 号梯 LEDg" )
   END_RUNG
   // the same network as SCL:
   IF "liftInfo".floor = "constant"."5楼" THEN
       "output"."1 号梯 LEDa" := TRUE;
       "output"."1 号梯 LEDb" := FALSE;
       "output"."1 号梯 LEDc" := TRUE;
       "output"."1 号梯 LEDd" := TRUE;
       "output"."1 号梯 LEDe" := FALSE;
       "output"."1 号梯 LEDf" := TRUE;
       "output"."1 号梯 LEDg" := TRUE;
   END_IF;
END_REGION

REGION Network 22: Six
   RUNG wire#powerrail
      { S7_Templates := "SrcType := UInt" } EQ_Contact(in1 := "liftInfo".floor, in2 := "constant"."6楼")
      wire#w1
      S_Coil( "output"."1 号梯 LEDa" )
   END_RUNG
   RUNG wire#w1
      R_Coil( "output"."1 号梯 LEDb" )
   END_RUNG
   RUNG wire#w1
      S_Coil( "output"."1 号梯 LEDc" )
   END_RUNG
   RUNG wire#w1
      S_Coil( "output"."1 号梯 LEDd" )
   END_RUNG
   RUNG wire#w1
      S_Coil( "output"."1 号梯 LEDe" )
   END_RUNG
   RUNG wire#w1
      S_Coil( "output"."1 号梯 LEDf" )
   END_RUNG
   RUNG wire#w1
      S_Coil( "output"."1 号梯 LEDg" )
   END_RUNG
   // the same network as SCL:
   IF "liftInfo".floor = "constant"."6楼" THEN
       "output"."1 号梯 LEDa" := TRUE;
       "output"."1 号梯 LEDb" := FALSE;
       "output"."1 号梯 LEDc" := TRUE;
       "output"."1 号梯 LEDd" := TRUE;
       "output"."1 号梯 LEDe" := TRUE;
       "output"."1 号梯 LEDf" := TRUE;
       "output"."1 号梯 LEDg" := TRUE;
   END_IF;
END_REGION
END_FUNCTION_BLOCK

FUNCTION_BLOCK "电梯上下行控制"   // FB2, LAD
{ S7_Optimized_Access := 'TRUE' }
VERSION : 0.1
   VAR
      上行开始 : Bool;
      登记 : Byte;
      下行开始 : Bool;
      反序楼层 : UInt;
      当前楼层 : Byte;
      上升层数 : UInt;
      下行层数 : UInt;
      firstStart : Bool;
   END_VAR
   VAR_TEMP
      tmp1 : Byte;
      tmp2 : Byte;
      tmp3 : UInt;
      tmp4 : UInt;
   END_VAR
   VAR_TEMP   // added for the SCL form of the ladder/FBD networks
      _w1 : Bool;
      _w2 : Bool;
   END_VAR
BEGIN

REGION Network 1
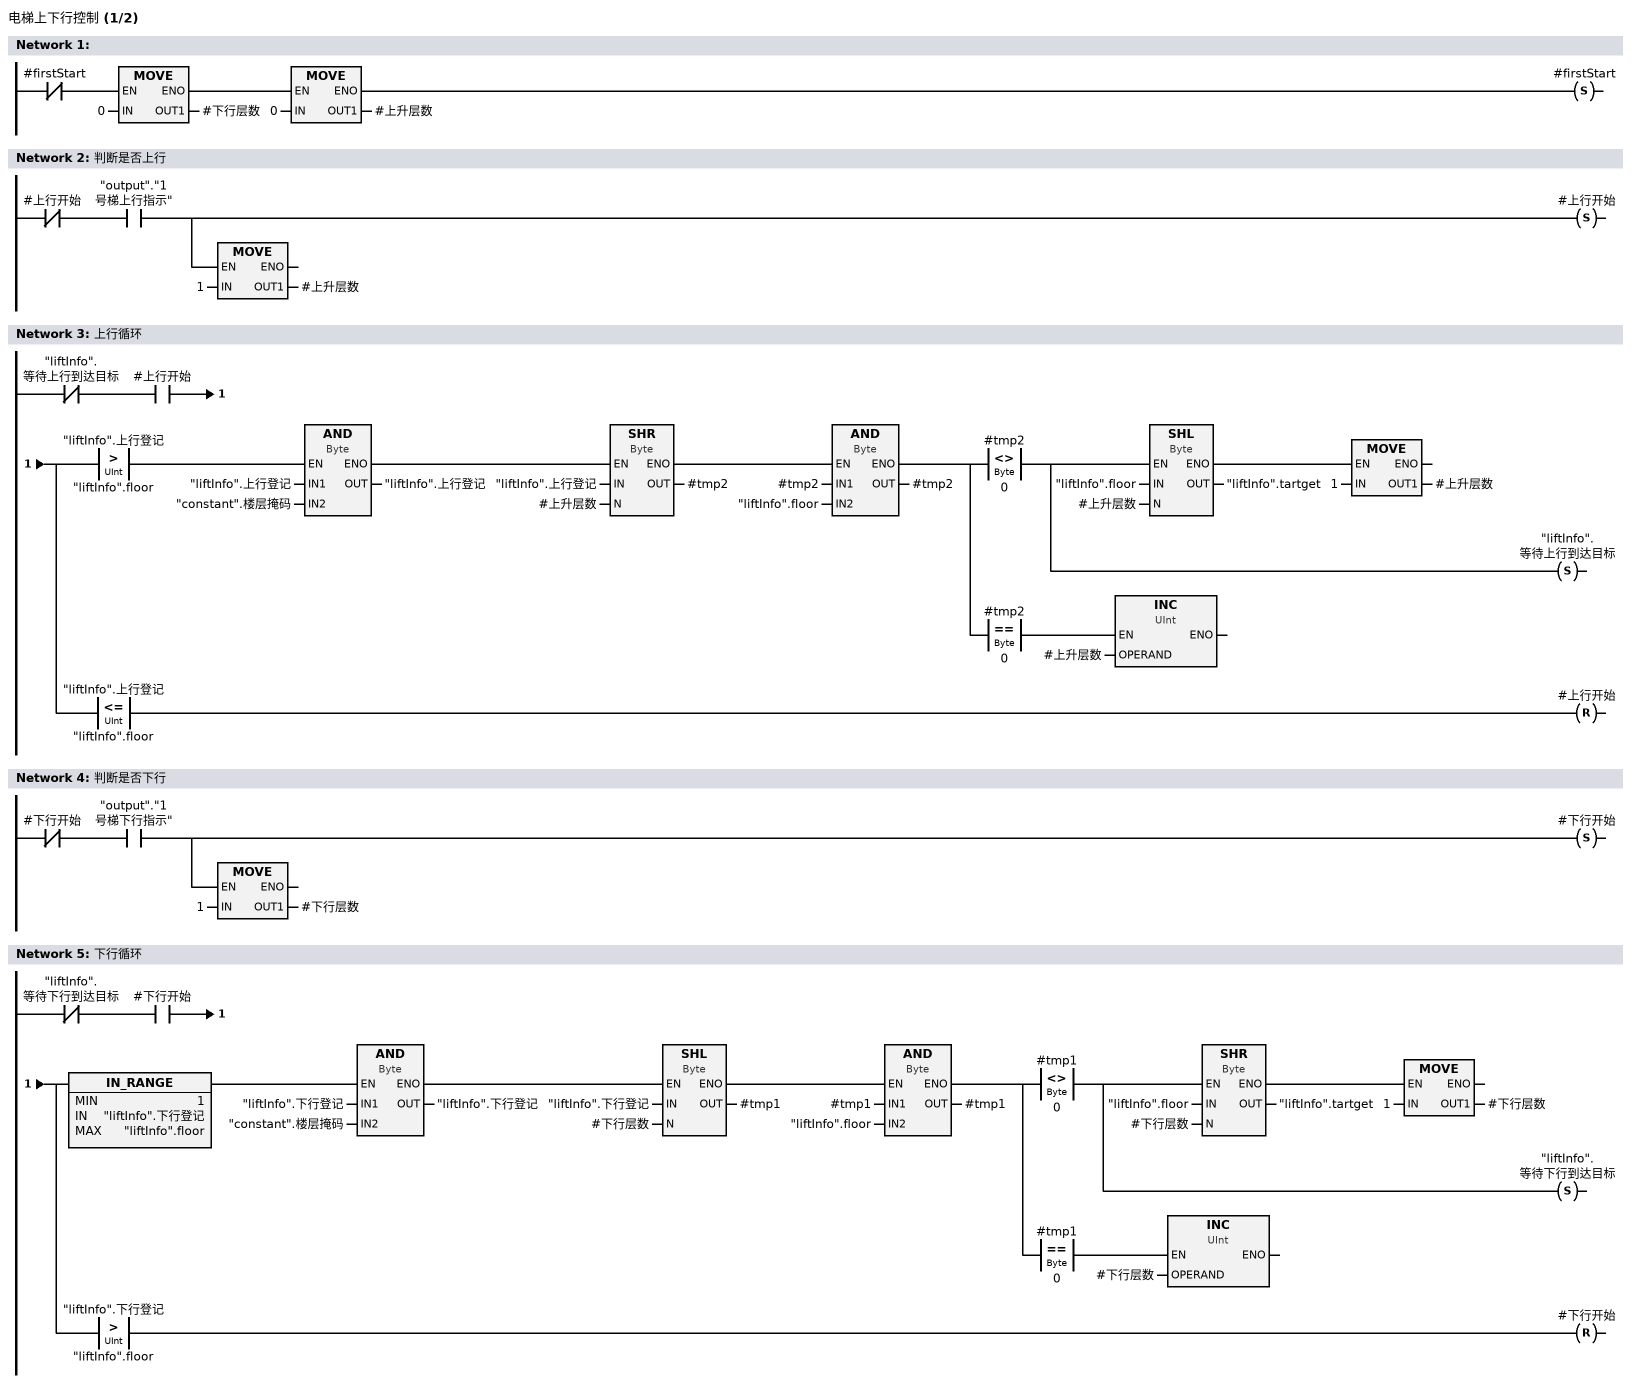
   RUNG wire#powerrail
      I_Contact( #firstStart )
      Move(in := 0, out1 => #下行层数)
      Move(in := 0, out1 => #上升层数)
      S_Coil( #firstStart )
   END_RUNG
   // the same network as SCL:
   IF NOT #firstStart THEN
       #下行层数 := 0;
       #上升层数 := 0;
       #firstStart := TRUE;
   END_IF;
END_REGION

REGION Network 2: 判断是否上行
   RUNG wire#powerrail
      I_Contact( #上行开始 )
      Contact( "output"."1 号梯上行指示" )
      wire#w1
      S_Coil( #上行开始 )
   END_RUNG
   RUNG wire#w1
      Move(in := 1, out1 => #上升层数)
   END_RUNG
   // the same network as SCL:
   #_w1 := NOT #上行开始 AND "output"."1 号梯上行指示";
   IF #_w1 THEN
       #上行开始 := TRUE;
       #上升层数 := 1;
   END_IF;
END_REGION

REGION Network 3: 上行循环
   RUNG wire#powerrail
      I_Contact( "liftInfo".等待上行到达目标 )
      Contact( #上行开始 )
      wire#w1
      { S7_Templates := "SrcType := UInt" } GT_Contact(in1 := "liftInfo".上行登记, in2 := "liftInfo".floor)
      { S7_Templates := "SrcType := Byte" } And(in1 := "liftInfo".上行登记, in2 := "constant".楼层掩码, out => "liftInfo".上行登记)
      { S7_Templates := "SrcType := Byte" } Shr(in := "liftInfo".上行登记, n := #上升层数, out => #tmp2)
      { S7_Templates := "SrcType := Byte" } And(in1 := #tmp2, in2 := "liftInfo".floor, out => #tmp2)
      wire#w2
      { S7_Templates := "SrcType := Byte" } NE_Contact(in1 := #tmp2, in2 := 0)
      wire#w3
      { S7_Templates := "SrcType := Byte" } Shl(in := "liftInfo".floor, n := #上升层数, out => "liftInfo".tartget)
      Move(in := 1, out1 => #上升层数)
   END_RUNG
   RUNG wire#w3
      S_Coil( "liftInfo".等待上行到达目标 )
   END_RUNG
   RUNG wire#w2
      { S7_Templates := "SrcType := Byte" } EQ_Contact(in1 := #tmp2, in2 := 0)
      { S7_Templates := "DestType := UInt" } Inc( #上升层数 )
   END_RUNG
   RUNG wire#w1
      { S7_Templates := "SrcType := UInt" } LE_Contact(in1 := "liftInfo".上行登记, in2 := "liftInfo".floor)
      R_Coil( #上行开始 )
   END_RUNG
   // the same network as SCL:
   #_w1 := NOT "liftInfo".等待上行到达目标 AND #上行开始;
   #_w2 := #_w1 AND ("liftInfo".上行登记 > "liftInfo".floor);
   IF #_w2 THEN
       "liftInfo".上行登记 := "liftInfo".上行登记 AND "constant".楼层掩码;
       #tmp2 := SHR(IN := "liftInfo".上行登记, N := #上升层数);
       #tmp2 := #tmp2 AND "liftInfo".floor;
   END_IF;
   IF #_w2 AND (#tmp2 <> 0) THEN
       "liftInfo".tartget := SHL(IN := "liftInfo".floor, N := #上升层数);
       #上升层数 := 1;
       "liftInfo".等待上行到达目标 := TRUE;
   END_IF;
   IF #_w2 AND (#tmp2 = 0) THEN #上升层数 := #上升层数 + 1; END_IF;
   IF #_w1 AND ("liftInfo".上行登记 <= "liftInfo".floor) THEN #上行开始 := FALSE; END_IF;
END_REGION

REGION Network 4: 判断是否下行
   RUNG wire#powerrail
      I_Contact( #下行开始 )
      Contact( "output"."1 号梯下行指示" )
      wire#w1
      S_Coil( #下行开始 )
   END_RUNG
   RUNG wire#w1
      Move(in := 1, out1 => #下行层数)
   END_RUNG
   // the same network as SCL:
   #_w1 := NOT #下行开始 AND "output"."1 号梯下行指示";
   IF #_w1 THEN
       #下行开始 := TRUE;
       #下行层数 := 1;
   END_IF;
END_REGION

REGION Network 5: 下行循环
   RUNG wire#powerrail
      I_Contact( "liftInfo".等待下行到达目标 )
      Contact( #下行开始 )
      wire#w1
      { S7_Templates := "SrcType := UInt" } InRange(min := 1, in := "liftInfo".下行登记, max := "liftInfo".floor)
      { S7_Templates := "SrcType := Byte" } And(in1 := "liftInfo".下行登记, in2 := "constant".楼层掩码, out => "liftInfo".下行登记)
      { S7_Templates := "SrcType := Byte" } Shl(in := "liftInfo".下行登记, n := #下行层数, out => #tmp1)
      { S7_Templates := "SrcType := Byte" } And(in1 := #tmp1, in2 := "liftInfo".floor, out => #tmp1)
      wire#w2
      { S7_Templates := "SrcType := Byte" } NE_Contact(in1 := #tmp1, in2 := 0)
      wire#w3
      { S7_Templates := "SrcType := Byte" } Shr(in := "liftInfo".floor, n := #下行层数, out => "liftInfo".tartget)
      Move(in := 1, out1 => #下行层数)
   END_RUNG
   RUNG wire#w3
      S_Coil( "liftInfo".等待下行到达目标 )
   END_RUNG
   RUNG wire#w2
      { S7_Templates := "SrcType := Byte" } EQ_Contact(in1 := #tmp1, in2 := 0)
      { S7_Templates := "DestType := UInt" } Inc( #下行层数 )
   END_RUNG
   RUNG wire#w1
      { S7_Templates := "SrcType := UInt" } GT_Contact(in1 := "liftInfo".下行登记, in2 := "liftInfo".floor)
      R_Coil( #下行开始 )
   END_RUNG
   // the same network as SCL:
   #_w1 := NOT "liftInfo".等待下行到达目标 AND #下行开始;
   #_w2 := #_w1 AND (1 <= "liftInfo".下行登记) AND ("liftInfo".下行登记 <= "liftInfo".floor);
   IF #_w2 THEN
       "liftInfo".下行登记 := "liftInfo".下行登记 AND "constant".楼层掩码;
       #tmp1 := SHL(IN := "liftInfo".下行登记, N := #下行层数);
       #tmp1 := #tmp1 AND "liftInfo".floor;
   END_IF;
   IF #_w2 AND (#tmp1 <> 0) THEN
       "liftInfo".tartget := SHR(IN := "liftInfo".floor, N := #下行层数);
       #下行层数 := 1;
       "liftInfo".等待下行到达目标 := TRUE;
   END_IF;
   IF #_w2 AND (#tmp1 = 0) THEN #下行层数 := #下行层数 + 1; END_IF;
   IF #_w1 AND ("liftInfo".下行登记 > "liftInfo".floor) THEN #下行开始 := FALSE; END_IF;
END_REGION

REGION Network 6: 静止时，判断上下行
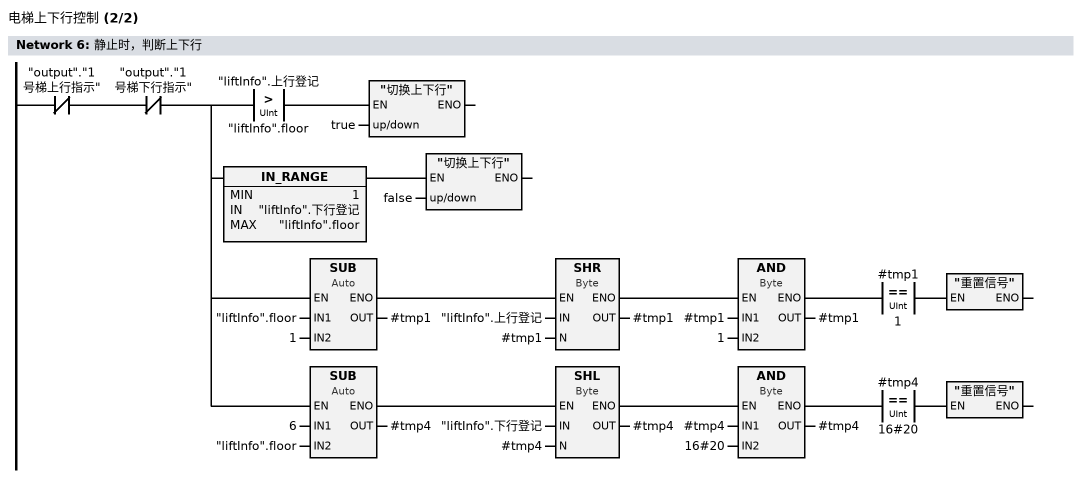
   RUNG wire#powerrail
      I_Contact( "output"."1 号梯上行指示" )
      I_Contact( "output"."1 号梯下行指示" )
      wire#w1
      { S7_Templates := "SrcType := UInt" } GT_Contact(in1 := "liftInfo".上行登记, in2 := "liftInfo".floor)
      "切换上下行"("up/down" := true)
   END_RUNG
   RUNG wire#w1
      { S7_Templates := "SrcType := UInt" } InRange(min := 1, in := "liftInfo".下行登记, max := "liftInfo".floor)
      "切换上下行"("up/down" := false)
   END_RUNG
   RUNG wire#w1
      Sub(in1 := "liftInfo".floor, in2 := 1, out => #tmp1)
      { S7_Templates := "SrcType := Byte" } Shr(in := "liftInfo".上行登记, n := #tmp1, out => #tmp1)
      { S7_Templates := "SrcType := Byte" } And(in1 := #tmp1, in2 := 1, out => #tmp1)
      { S7_Templates := "SrcType := UInt" } EQ_Contact(in1 := #tmp1, in2 := 1)
      "重置信号"()
   END_RUNG
   RUNG wire#w1
      Sub(in1 := 6, in2 := "liftInfo".floor, out => #tmp4)
      { S7_Templates := "SrcType := Byte" } Shl(in := "liftInfo".下行登记, n := #tmp4, out => #tmp4)
      { S7_Templates := "SrcType := Byte" } And(in1 := #tmp4, in2 := 16#20, out => #tmp4)
      { S7_Templates := "SrcType := UInt" } EQ_Contact(in1 := #tmp4, in2 := 16#20)
      "重置信号"()
   END_RUNG
   // the same network as SCL:
   #_w1 := NOT "output"."1 号梯上行指示" AND NOT "output"."1 号梯下行指示";
   IF #_w1 AND ("liftInfo".上行登记 > "liftInfo".floor) THEN "切换上下行"("up/down" := true); END_IF;
   IF #_w1 AND (1 <= "liftInfo".下行登记) AND ("liftInfo".下行登记 <= "liftInfo".floor) THEN
       "切换上下行"("up/down" := false);
   END_IF;
   IF #_w1 THEN
       #tmp1 := "liftInfo".floor - 1;
       #tmp1 := SHR(IN := "liftInfo".上行登记, N := #tmp1);
       #tmp1 := #tmp1 AND 1;
   END_IF;
   IF #_w1 AND (#tmp1 = 1) THEN "重置信号"(); END_IF;
   IF #_w1 THEN
       #tmp4 := 6 - "liftInfo".floor;
       #tmp4 := SHL(IN := "liftInfo".下行登记, N := #tmp4);
       #tmp4 := #tmp4 AND 16#20;
   END_IF;
   IF #_w1 AND (#tmp4 = 16#20) THEN "重置信号"(); END_IF;
END_REGION
END_FUNCTION_BLOCK

FUNCTION_BLOCK "错误检测"   // FB3, LAD
{ S7_Optimized_Access := 'TRUE' }
VERSION : 0.1
   VAR_TEMP   // added for the SCL form of the ladder/FBD networks
      _w1 : Bool;
   END_VAR
BEGIN

REGION Network 1
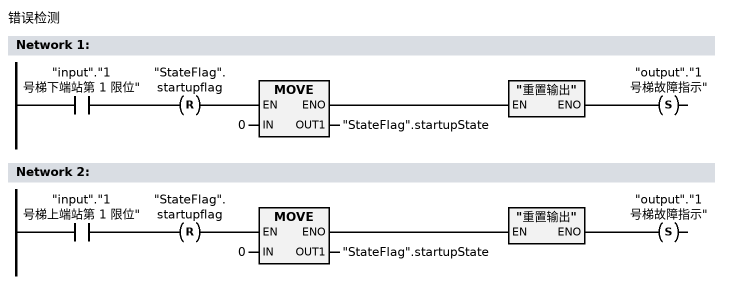
   RUNG wire#powerrail
      Contact( "input"."1 号梯下端站第 1 限位" )
      R_Coil( "StateFlag".startupflag )
      Move(in := 0, out1 => "StateFlag".startupState)
      "重置输出"()
      S_Coil( "output"."1 号梯故障指示" )
   END_RUNG
   // the same network as SCL:
   IF "input"."1 号梯下端站第 1 限位" THEN
       "StateFlag".startupflag := FALSE;
       "StateFlag".startupState := 0;
   END_IF;
   "重置输出"(EN := "input"."1 号梯下端站第 1 限位", ENO => #_w1);
   IF #_w1 THEN "output"."1 号梯故障指示" := TRUE; END_IF;
END_REGION

REGION Network 2
   RUNG wire#powerrail
      Contact( "input"."1 号梯上端站第 1 限位" )
      R_Coil( "StateFlag".startupflag )
      Move(in := 0, out1 => "StateFlag".startupState)
      "重置输出"()
      S_Coil( "output"."1 号梯故障指示" )
   END_RUNG
   // the same network as SCL:
   IF "input"."1 号梯上端站第 1 限位" THEN
       "StateFlag".startupflag := FALSE;
       "StateFlag".startupState := 0;
   END_IF;
   "重置输出"(EN := "input"."1 号梯上端站第 1 限位", ENO => #_w1);
   IF #_w1 THEN "output"."1 号梯故障指示" := TRUE; END_IF;
END_REGION
END_FUNCTION_BLOCK

FUNCTION_BLOCK "开关门"   // FB4, LAD
{ S7_Optimized_Access := 'TRUE' }
VERSION : 0.1
   VAR_TEMP   // added for the SCL form of the ladder/FBD networks
      _w1 : Bool;
      _w2 : Bool;
   END_VAR
BEGIN

REGION Network 1: 按键开门
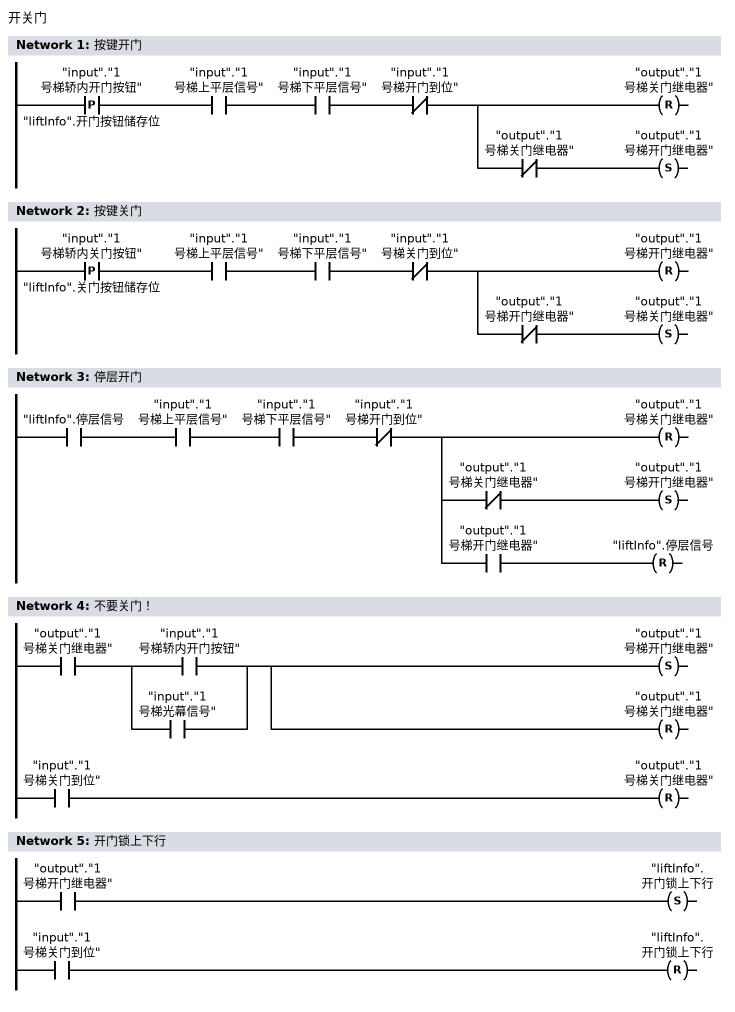
   RUNG wire#powerrail
      P_Contact(operand := "input"."1 号梯轿内开门按钮", bit := "liftInfo".开门按钮储存位)
      Contact( "input"."1 号梯上平层信号" )
      Contact( "input"."1 号梯下平层信号" )
      I_Contact( "input"."1 号梯开门到位" )
      wire#w1
      R_Coil( "output"."1 号梯关门继电器" )
   END_RUNG
   RUNG wire#w1
      I_Contact( "output"."1 号梯关门继电器" )
      S_Coil( "output"."1 号梯开门继电器" )
   END_RUNG
   // the same network as SCL:
   #_w1 := "input"."1 号梯轿内开门按钮" AND NOT "liftInfo".开门按钮储存位;   // rising edge of "input"."1 号梯轿内开门按钮"
   "liftInfo".开门按钮储存位 := "input"."1 号梯轿内开门按钮";
   #_w2 := #_w1 AND "input"."1 号梯上平层信号" AND "input"."1 号梯下平层信号" AND NOT "input"."1 号梯开门到位";
   IF #_w2 THEN "output"."1 号梯关门继电器" := FALSE; END_IF;
   IF #_w2 AND NOT "output"."1 号梯关门继电器" THEN "output"."1 号梯开门继电器" := TRUE; END_IF;
END_REGION

REGION Network 2: 按键关门
   RUNG wire#powerrail
      P_Contact(operand := "input"."1 号梯轿内关门按钮", bit := "liftInfo".关门按钮储存位)
      Contact( "input"."1 号梯上平层信号" )
      Contact( "input"."1 号梯下平层信号" )
      I_Contact( "input"."1 号梯关门到位" )
      wire#w1
      R_Coil( "output"."1 号梯开门继电器" )
   END_RUNG
   RUNG wire#w1
      I_Contact( "output"."1 号梯开门继电器" )
      S_Coil( "output"."1 号梯关门继电器" )
   END_RUNG
   // the same network as SCL:
   #_w1 := "input"."1 号梯轿内关门按钮" AND NOT "liftInfo".关门按钮储存位;   // rising edge of "input"."1 号梯轿内关门按钮"
   "liftInfo".关门按钮储存位 := "input"."1 号梯轿内关门按钮";
   #_w2 := #_w1 AND "input"."1 号梯上平层信号" AND "input"."1 号梯下平层信号" AND NOT "input"."1 号梯关门到位";
   IF #_w2 THEN "output"."1 号梯开门继电器" := FALSE; END_IF;
   IF #_w2 AND NOT "output"."1 号梯开门继电器" THEN "output"."1 号梯关门继电器" := TRUE; END_IF;
END_REGION

REGION Network 3: 停层开门
   RUNG wire#powerrail
      Contact( "liftInfo".停层信号 )
      Contact( "input"."1 号梯上平层信号" )
      Contact( "input"."1 号梯下平层信号" )
      I_Contact( "input"."1 号梯开门到位" )
      wire#w1
      R_Coil( "output"."1 号梯关门继电器" )
   END_RUNG
   RUNG wire#w1
      I_Contact( "output"."1 号梯关门继电器" )
      S_Coil( "output"."1 号梯开门继电器" )
   END_RUNG
   RUNG wire#w1
      Contact( "output"."1 号梯开门继电器" )
      R_Coil( "liftInfo".停层信号 )
   END_RUNG
   // the same network as SCL:
   #_w1 := "liftInfo".停层信号 AND "input"."1 号梯上平层信号" AND "input"."1 号梯下平层信号" AND NOT "input"."1 号梯开门到位";
   IF #_w1 THEN "output"."1 号梯关门继电器" := FALSE; END_IF;
   IF #_w1 AND NOT "output"."1 号梯关门继电器" THEN "output"."1 号梯开门继电器" := TRUE; END_IF;
   IF #_w1 AND "output"."1 号梯开门继电器" THEN "liftInfo".停层信号 := FALSE; END_IF;
END_REGION

REGION Network 4: 不要关门！
   RUNG wire#powerrail
      Contact( "output"."1 号梯关门继电器" )
      wire#w1
      Contact( "input"."1 号梯轿内开门按钮" )
      wire#w2
      S_Coil( "output"."1 号梯开门继电器" )
   END_RUNG
   RUNG wire#w1
      Contact( "input"."1 号梯光幕信号" )
   END_RUNG wire#w2
   RUNG wire#w2
      R_Coil( "output"."1 号梯关门继电器" )
   END_RUNG
   RUNG wire#powerrail
      Contact( "input"."1 号梯关门到位" )
      R_Coil( "output"."1 号梯关门继电器" )
   END_RUNG
   // the same network as SCL:
   IF "output"."1 号梯关门继电器" AND ("input"."1 号梯轿内开门按钮" OR "input"."1 号梯光幕信号") THEN
       "output"."1 号梯开门继电器" := TRUE;
       "output"."1 号梯关门继电器" := FALSE;
   END_IF;
   IF "input"."1 号梯关门到位" THEN "output"."1 号梯关门继电器" := FALSE; END_IF;
END_REGION

REGION Network 5: 开门锁上下行
   RUNG wire#powerrail
      Contact( "output"."1 号梯开门继电器" )
      S_Coil( "liftInfo".开门锁上下行 )
   END_RUNG
   RUNG wire#powerrail
      Contact( "input"."1 号梯关门到位" )
      R_Coil( "liftInfo".开门锁上下行 )
   END_RUNG
   // the same network as SCL:
   IF "output"."1 号梯开门继电器" THEN "liftInfo".开门锁上下行 := TRUE; END_IF;
   IF "input"."1 号梯关门到位" THEN "liftInfo".开门锁上下行 := FALSE; END_IF;
END_REGION
END_FUNCTION_BLOCK

FUNCTION "赋值数据" : Void   // FC1, LAD
{ S7_Optimized_Access := 'TRUE' }
VERSION : 0.1
   VAR_INPUT
      类型 : UInt;
      位数 : UInt;
      "置位/复位" : Bool;
   END_VAR
   VAR_TEMP
      tmp1 : Byte;
   END_VAR
   VAR_TEMP   // added for the SCL form of the ladder/FBD networks
      _w1 : Bool;
   END_VAR
BEGIN

REGION Network 1: 梯内按钮输入
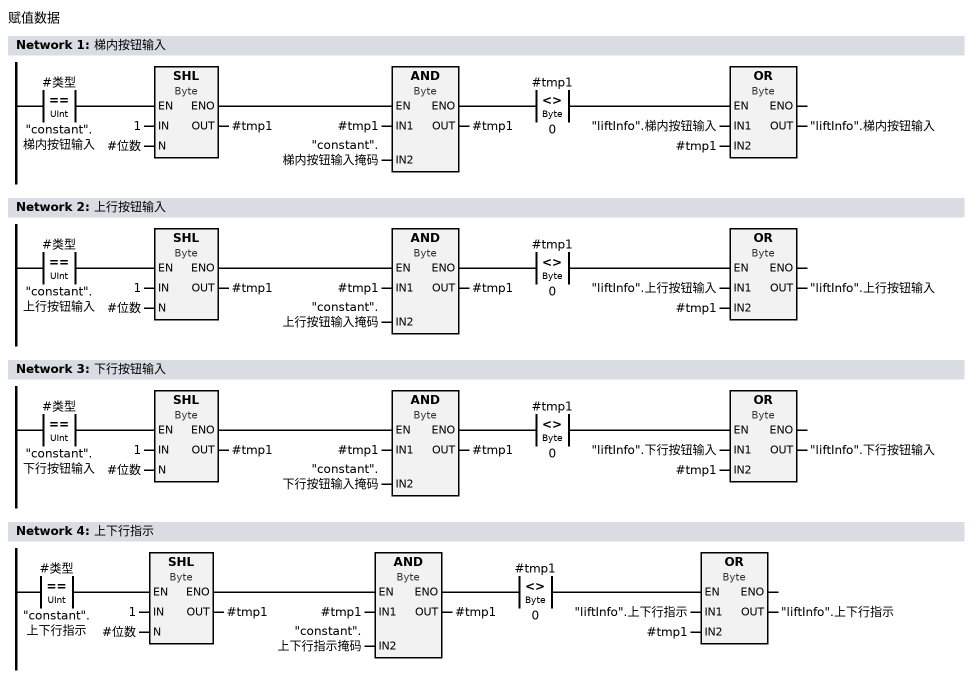
   #_w1 := #类型 = "constant".梯内按钮输入;
   IF #_w1 THEN
       #tmp1 := SHL(IN := 1, N := #位数);
       #tmp1 := #tmp1 AND "constant".梯内按钮输入掩码;
   END_IF;
   IF #_w1 AND (#tmp1 <> 0) THEN "liftInfo".梯内按钮输入 := "liftInfo".梯内按钮输入 OR #tmp1; END_IF;
END_REGION

REGION Network 2: 上行按钮输入
   #_w1 := #类型 = "constant".上行按钮输入;
   IF #_w1 THEN
       #tmp1 := SHL(IN := 1, N := #位数);
       #tmp1 := #tmp1 AND "constant".上行按钮输入掩码;
   END_IF;
   IF #_w1 AND (#tmp1 <> 0) THEN "liftInfo".上行按钮输入 := "liftInfo".上行按钮输入 OR #tmp1; END_IF;
END_REGION

REGION Network 3: 下行按钮输入
   #_w1 := #类型 = "constant".下行按钮输入;
   IF #_w1 THEN
       #tmp1 := SHL(IN := 1, N := #位数);
       #tmp1 := #tmp1 AND "constant".下行按钮输入掩码;
   END_IF;
   IF #_w1 AND (#tmp1 <> 0) THEN "liftInfo".下行按钮输入 := "liftInfo".下行按钮输入 OR #tmp1; END_IF;
END_REGION

REGION Network 4: 上下行指示
   #_w1 := #类型 = "constant".上下行指示;
   IF #_w1 THEN
       #tmp1 := SHL(IN := 1, N := #位数);
       #tmp1 := #tmp1 AND "constant".上下行指示掩码;
   END_IF;
   IF #_w1 AND (#tmp1 <> 0) THEN "liftInfo".上下行指示 := "liftInfo".上下行指示 OR #tmp1; END_IF;
END_REGION
END_FUNCTION

FUNCTION "切换上下行" : Void   // FC2, LAD
{ S7_Optimized_Access := 'TRUE' }
VERSION : 0.1
   VAR_INPUT
      "up/down" : Bool;   // 上行为1,下行为0
   END_VAR
BEGIN

REGION Network 1
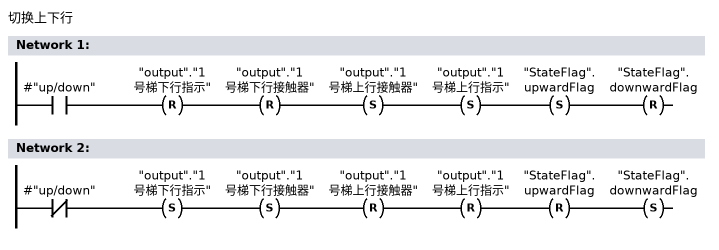
   RUNG wire#powerrail
      Contact( #"up/down" )
      R_Coil( "output"."1 号梯下行指示" )
      R_Coil( "output"."1 号梯下行接触器" )
      S_Coil( "output"."1 号梯上行接触器" )
      S_Coil( "output"."1 号梯上行指示" )
      S_Coil( "StateFlag".upwardFlag )
      R_Coil( "StateFlag".downwardFlag )
   END_RUNG
   // the same network as SCL:
   IF #"up/down" THEN
       "output"."1 号梯下行指示" := FALSE;
       "output"."1 号梯下行接触器" := FALSE;
       "output"."1 号梯上行接触器" := TRUE;
       "output"."1 号梯上行指示" := TRUE;
       "StateFlag".upwardFlag := TRUE;
       "StateFlag".downwardFlag := FALSE;
   END_IF;
END_REGION

REGION Network 2
   RUNG wire#powerrail
      I_Contact( #"up/down" )
      S_Coil( "output"."1 号梯下行指示" )
      S_Coil( "output"."1 号梯下行接触器" )
      R_Coil( "output"."1 号梯上行接触器" )
      R_Coil( "output"."1 号梯上行指示" )
      R_Coil( "StateFlag".upwardFlag )
      S_Coil( "StateFlag".downwardFlag )
   END_RUNG
   // the same network as SCL:
   IF NOT #"up/down" THEN
       "output"."1 号梯下行指示" := TRUE;
       "output"."1 号梯下行接触器" := TRUE;
       "output"."1 号梯上行接触器" := FALSE;
       "output"."1 号梯上行指示" := FALSE;
       "StateFlag".upwardFlag := FALSE;
       "StateFlag".downwardFlag := TRUE;
   END_IF;
END_REGION
END_FUNCTION

FUNCTION "重置制动器" : Void   // FC3, LAD
{ S7_Optimized_Access := 'TRUE' }
VERSION : 0.1
BEGIN

REGION Network 1
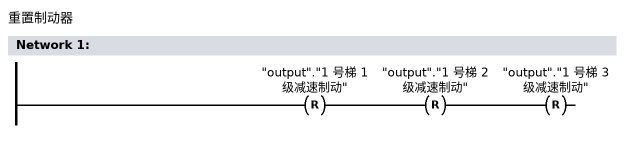
   RUNG wire#powerrail
      R_Coil( "output"."1 号梯 1 级减速制动" )
      R_Coil( "output"."1 号梯 2 级减速制动" )
      R_Coil( "output"."1 号梯 3 级减速制动" )
   END_RUNG
   // the same network as SCL:
   "output"."1 号梯 1 级减速制动" := FALSE;
   "output"."1 号梯 2 级减速制动" := FALSE;
   "output"."1 号梯 3 级减速制动" := FALSE;
END_REGION
END_FUNCTION

FUNCTION "重置上下行" : Void   // FC4, LAD
{ S7_Optimized_Access := 'TRUE' }
VERSION : 0.1
BEGIN

REGION Network 1
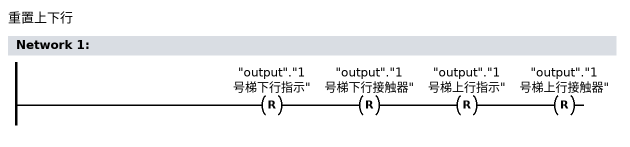
   RUNG wire#powerrail
      R_Coil( "output"."1 号梯下行指示" )
      R_Coil( "output"."1 号梯下行接触器" )
      R_Coil( "output"."1 号梯上行指示" )
      R_Coil( "output"."1 号梯上行接触器" )
   END_RUNG
   // the same network as SCL:
   "output"."1 号梯下行指示" := FALSE;
   "output"."1 号梯下行接触器" := FALSE;
   "output"."1 号梯上行指示" := FALSE;
   "output"."1 号梯上行接触器" := FALSE;
END_REGION
END_FUNCTION

FUNCTION "获取数据" : Void   // FC5, LAD
{ S7_Optimized_Access := 'TRUE' }
VERSION : 0.1
   VAR_INPUT
      类型 : UInt;
      位数 : UInt;
   END_VAR
   VAR_OUTPUT
      数据 : Bool;
   END_VAR
   VAR_TEMP
      tmp1 : Byte;
   END_VAR
   VAR_TEMP   // added for the SCL form of the ladder/FBD networks
      _w1 : Bool;
   END_VAR
BEGIN

REGION Network 1: 梯内按钮输入
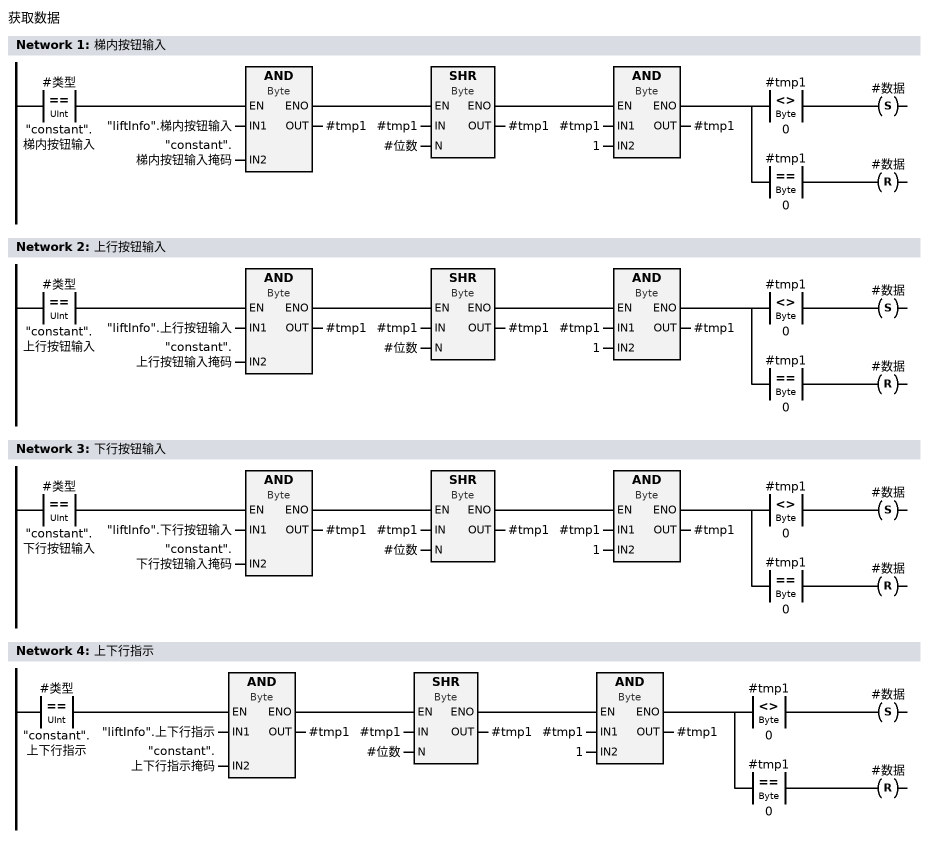
   RUNG wire#powerrail
      { S7_Templates := "SrcType := UInt" } EQ_Contact(in1 := #类型, in2 := "constant".梯内按钮输入)
      { S7_Templates := "SrcType := Byte" } And(in1 := "liftInfo".梯内按钮输入, in2 := "constant".梯内按钮输入掩码, out => #tmp1)
      { S7_Templates := "SrcType := Byte" } Shr(in := #tmp1, n := #位数, out => #tmp1)
      { S7_Templates := "SrcType := Byte" } And(in1 := #tmp1, in2 := 1, out => #tmp1)
      wire#w1
      { S7_Templates := "SrcType := Byte" } NE_Contact(in1 := #tmp1, in2 := 0)
      S_Coil( #数据 )
   END_RUNG
   RUNG wire#w1
      { S7_Templates := "SrcType := Byte" } EQ_Contact(in1 := #tmp1, in2 := 0)
      R_Coil( #数据 )
   END_RUNG
   // the same network as SCL:
   #_w1 := #类型 = "constant".梯内按钮输入;
   IF #_w1 THEN
       #tmp1 := "liftInfo".梯内按钮输入 AND "constant".梯内按钮输入掩码;
       #tmp1 := SHR(IN := #tmp1, N := #位数);
       #tmp1 := #tmp1 AND 1;
   END_IF;
   IF #_w1 AND (#tmp1 <> 0) THEN #数据 := TRUE; END_IF;
   IF #_w1 AND (#tmp1 = 0) THEN #数据 := FALSE; END_IF;
END_REGION

REGION Network 2: 上行按钮输入
   RUNG wire#powerrail
      { S7_Templates := "SrcType := UInt" } EQ_Contact(in1 := #类型, in2 := "constant".上行按钮输入)
      { S7_Templates := "SrcType := Byte" } And(in1 := "liftInfo".上行按钮输入, in2 := "constant".上行按钮输入掩码, out => #tmp1)
      { S7_Templates := "SrcType := Byte" } Shr(in := #tmp1, n := #位数, out => #tmp1)
      { S7_Templates := "SrcType := Byte" } And(in1 := #tmp1, in2 := 1, out => #tmp1)
      wire#w1
      { S7_Templates := "SrcType := Byte" } NE_Contact(in1 := #tmp1, in2 := 0)
      S_Coil( #数据 )
   END_RUNG
   RUNG wire#w1
      { S7_Templates := "SrcType := Byte" } EQ_Contact(in1 := #tmp1, in2 := 0)
      R_Coil( #数据 )
   END_RUNG
   // the same network as SCL:
   #_w1 := #类型 = "constant".上行按钮输入;
   IF #_w1 THEN
       #tmp1 := "liftInfo".上行按钮输入 AND "constant".上行按钮输入掩码;
       #tmp1 := SHR(IN := #tmp1, N := #位数);
       #tmp1 := #tmp1 AND 1;
   END_IF;
   IF #_w1 AND (#tmp1 <> 0) THEN #数据 := TRUE; END_IF;
   IF #_w1 AND (#tmp1 = 0) THEN #数据 := FALSE; END_IF;
END_REGION

REGION Network 3: 下行按钮输入
   RUNG wire#powerrail
      { S7_Templates := "SrcType := UInt" } EQ_Contact(in1 := #类型, in2 := "constant".下行按钮输入)
      { S7_Templates := "SrcType := Byte" } And(in1 := "liftInfo".下行按钮输入, in2 := "constant".下行按钮输入掩码, out => #tmp1)
      { S7_Templates := "SrcType := Byte" } Shr(in := #tmp1, n := #位数, out => #tmp1)
      { S7_Templates := "SrcType := Byte" } And(in1 := #tmp1, in2 := 1, out => #tmp1)
      wire#w1
      { S7_Templates := "SrcType := Byte" } NE_Contact(in1 := #tmp1, in2 := 0)
      S_Coil( #数据 )
   END_RUNG
   RUNG wire#w1
      { S7_Templates := "SrcType := Byte" } EQ_Contact(in1 := #tmp1, in2 := 0)
      R_Coil( #数据 )
   END_RUNG
   // the same network as SCL:
   #_w1 := #类型 = "constant".下行按钮输入;
   IF #_w1 THEN
       #tmp1 := "liftInfo".下行按钮输入 AND "constant".下行按钮输入掩码;
       #tmp1 := SHR(IN := #tmp1, N := #位数);
       #tmp1 := #tmp1 AND 1;
   END_IF;
   IF #_w1 AND (#tmp1 <> 0) THEN #数据 := TRUE; END_IF;
   IF #_w1 AND (#tmp1 = 0) THEN #数据 := FALSE; END_IF;
END_REGION

REGION Network 4: 上下行指示
   RUNG wire#powerrail
      { S7_Templates := "SrcType := UInt" } EQ_Contact(in1 := #类型, in2 := "constant".上下行指示)
      { S7_Templates := "SrcType := Byte" } And(in1 := "liftInfo".上下行指示, in2 := "constant".上下行指示掩码, out => #tmp1)
      { S7_Templates := "SrcType := Byte" } Shr(in := #tmp1, n := #位数, out => #tmp1)
      { S7_Templates := "SrcType := Byte" } And(in1 := #tmp1, in2 := 1, out => #tmp1)
      wire#w1
      { S7_Templates := "SrcType := Byte" } NE_Contact(in1 := #tmp1, in2 := 0)
      S_Coil( #数据 )
   END_RUNG
   RUNG wire#w1
      { S7_Templates := "SrcType := Byte" } EQ_Contact(in1 := #tmp1, in2 := 0)
      R_Coil( #数据 )
   END_RUNG
   // the same network as SCL:
   #_w1 := #类型 = "constant".上下行指示;
   IF #_w1 THEN
       #tmp1 := "liftInfo".上下行指示 AND "constant".上下行指示掩码;
       #tmp1 := SHR(IN := #tmp1, N := #位数);
       #tmp1 := #tmp1 AND 1;
   END_IF;
   IF #_w1 AND (#tmp1 <> 0) THEN #数据 := TRUE; END_IF;
   IF #_w1 AND (#tmp1 = 0) THEN #数据 := FALSE; END_IF;
END_REGION
END_FUNCTION

FUNCTION "重置信号" : Void   // FC6, LAD
{ S7_Optimized_Access := 'TRUE' }
VERSION : 0.1
   VAR_TEMP
      登记 : Byte;
      tmp1 : Byte;
   END_VAR
   VAR_TEMP   // added for the SCL form of the ladder/FBD networks
      _w1 : Bool;
      _w2 : Bool;
      _w3 : Bool;
   END_VAR
BEGIN

REGION Network 1
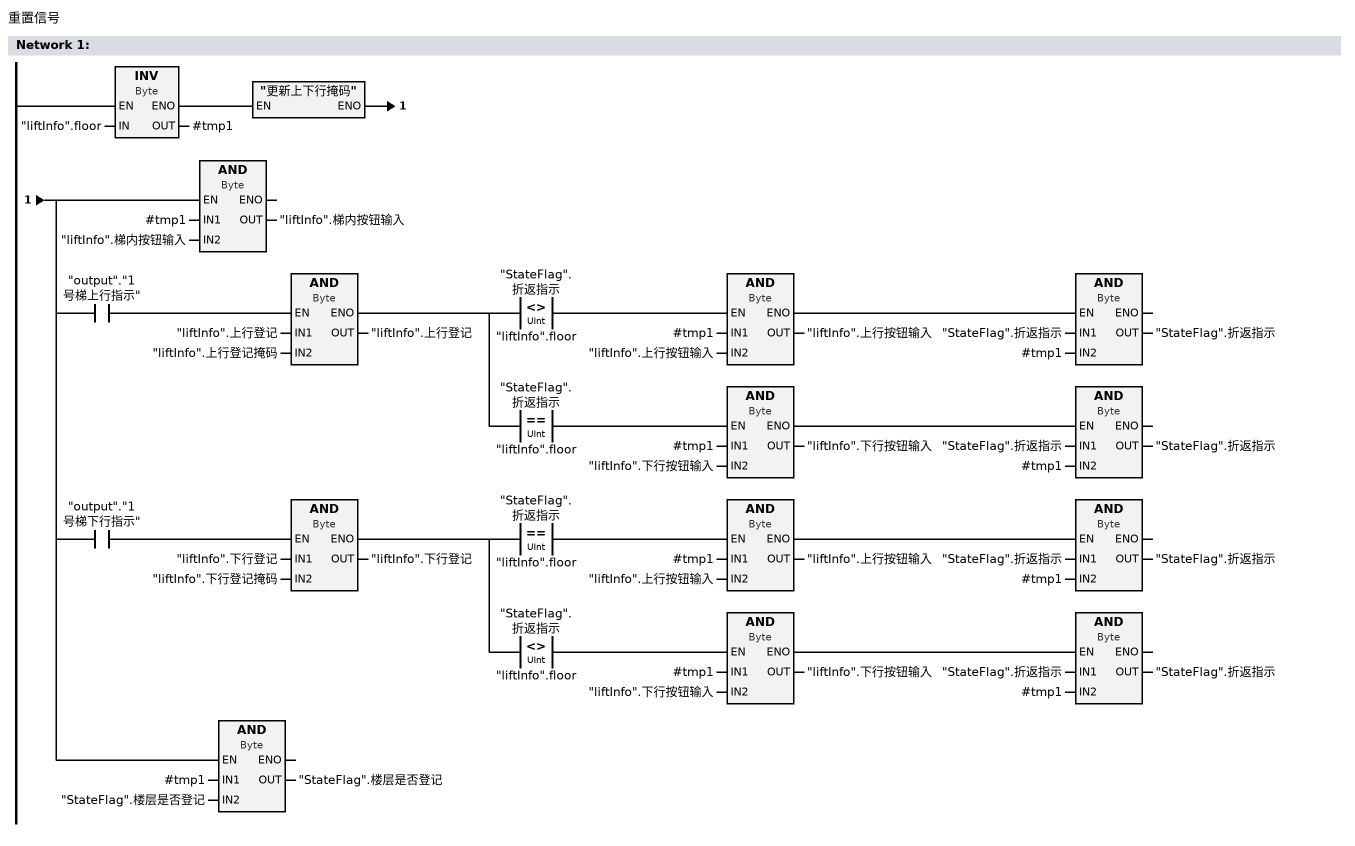
   RUNG wire#powerrail
      { S7_Templates := "SrcType := Byte" } Inv(in := "liftInfo".floor, out => #tmp1)
      "更新上下行掩码"()
      wire#w1
      { S7_Templates := "SrcType := Byte" } And(in1 := #tmp1, in2 := "liftInfo".梯内按钮输入, out => "liftInfo".梯内按钮输入)
   END_RUNG
   RUNG wire#w1
      Contact( "output"."1 号梯上行指示" )
      { S7_Templates := "SrcType := Byte" } And(in1 := "liftInfo".上行登记, in2 := "liftInfo".上行登记掩码, out => "liftInfo".上行登记)
      wire#w2
      { S7_Templates := "SrcType := UInt" } NE_Contact(in1 := "StateFlag".折返指示, in2 := "liftInfo".floor)
      { S7_Templates := "SrcType := Byte" } And(in1 := #tmp1, in2 := "liftInfo".上行按钮输入, out => "liftInfo".上行按钮输入)
      { S7_Templates := "SrcType := Byte" } And(in1 := "StateFlag".折返指示, in2 := #tmp1, out => "StateFlag".折返指示)
   END_RUNG
   RUNG wire#w2
      { S7_Templates := "SrcType := UInt" } EQ_Contact(in1 := "StateFlag".折返指示, in2 := "liftInfo".floor)
      { S7_Templates := "SrcType := Byte" } And(in1 := #tmp1, in2 := "liftInfo".下行按钮输入, out => "liftInfo".下行按钮输入)
      { S7_Templates := "SrcType := Byte" } And(in1 := "StateFlag".折返指示, in2 := #tmp1, out => "StateFlag".折返指示)
   END_RUNG
   RUNG wire#w1
      Contact( "output"."1 号梯下行指示" )
      { S7_Templates := "SrcType := Byte" } And(in1 := "liftInfo".下行登记, in2 := "liftInfo".下行登记掩码, out => "liftInfo".下行登记)
      wire#w3
      { S7_Templates := "SrcType := UInt" } EQ_Contact(in1 := "StateFlag".折返指示, in2 := "liftInfo".floor)
      { S7_Templates := "SrcType := Byte" } And(in1 := #tmp1, in2 := "liftInfo".上行按钮输入, out => "liftInfo".上行按钮输入)
      { S7_Templates := "SrcType := Byte" } And(in1 := "StateFlag".折返指示, in2 := #tmp1, out => "StateFlag".折返指示)
   END_RUNG
   RUNG wire#w3
      { S7_Templates := "SrcType := UInt" } NE_Contact(in1 := "StateFlag".折返指示, in2 := "liftInfo".floor)
      { S7_Templates := "SrcType := Byte" } And(in1 := #tmp1, in2 := "liftInfo".下行按钮输入, out => "liftInfo".下行按钮输入)
      { S7_Templates := "SrcType := Byte" } And(in1 := "StateFlag".折返指示, in2 := #tmp1, out => "StateFlag".折返指示)
   END_RUNG
   RUNG wire#w1
      { S7_Templates := "SrcType := Byte" } And(in1 := #tmp1, in2 := "StateFlag".楼层是否登记, out => "StateFlag".楼层是否登记)
   END_RUNG
   // the same network as SCL:
   #tmp1 := NOT "liftInfo".floor;
   "更新上下行掩码"(ENO => #_w1);
   IF #_w1 THEN "liftInfo".梯内按钮输入 := #tmp1 AND "liftInfo".梯内按钮输入; END_IF;
   #_w2 := #_w1 AND "output"."1 号梯上行指示";
   IF #_w2 THEN "liftInfo".上行登记 := "liftInfo".上行登记 AND "liftInfo".上行登记掩码; END_IF;
   IF #_w2 AND ("StateFlag".折返指示 <> "liftInfo".floor) THEN
       "liftInfo".上行按钮输入 := #tmp1 AND "liftInfo".上行按钮输入;
       "StateFlag".折返指示 := "StateFlag".折返指示 AND #tmp1;
   END_IF;
   IF #_w2 AND ("StateFlag".折返指示 = "liftInfo".floor) THEN
       "liftInfo".下行按钮输入 := #tmp1 AND "liftInfo".下行按钮输入;
       "StateFlag".折返指示 := "StateFlag".折返指示 AND #tmp1;
   END_IF;
   #_w3 := #_w1 AND "output"."1 号梯下行指示";
   IF #_w3 THEN "liftInfo".下行登记 := "liftInfo".下行登记 AND "liftInfo".下行登记掩码; END_IF;
   IF #_w3 AND ("StateFlag".折返指示 = "liftInfo".floor) THEN
       "liftInfo".上行按钮输入 := #tmp1 AND "liftInfo".上行按钮输入;
       "StateFlag".折返指示 := "StateFlag".折返指示 AND #tmp1;
   END_IF;
   IF #_w3 AND ("StateFlag".折返指示 <> "liftInfo".floor) THEN
       "liftInfo".下行按钮输入 := #tmp1 AND "liftInfo".下行按钮输入;
       "StateFlag".折返指示 := "StateFlag".折返指示 AND #tmp1;
   END_IF;
   IF #_w1 THEN "StateFlag".楼层是否登记 := #tmp1 AND "StateFlag".楼层是否登记; END_IF;
END_REGION
END_FUNCTION

FUNCTION "重置输出" : Void   // FC7, LAD
{ S7_Optimized_Access := 'TRUE' }
VERSION : 0.1
   VAR_TEMP   // added for the SCL form of the ladder/FBD networks
      _w1 : Bool;
   END_VAR
BEGIN

REGION Network 1
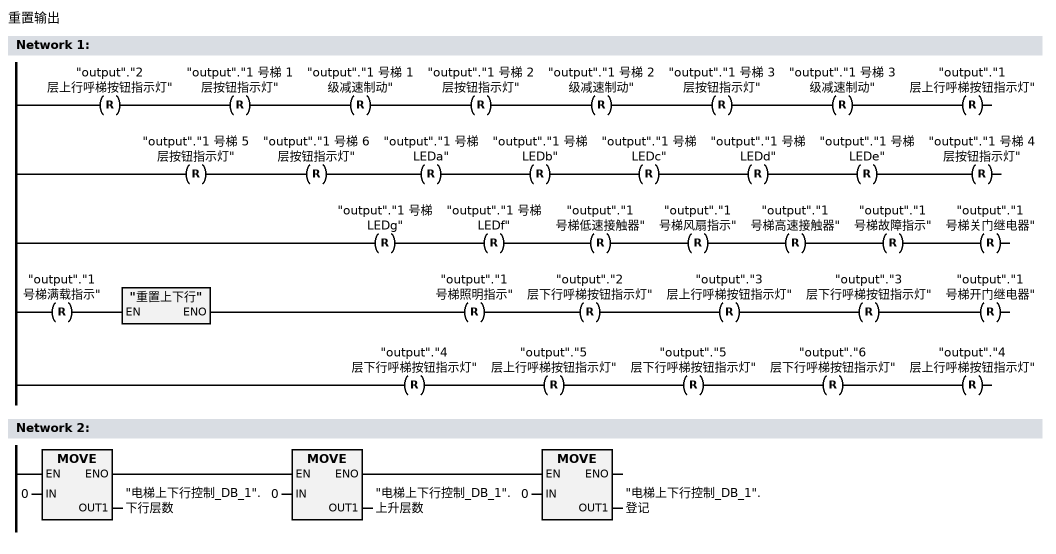
   RUNG wire#powerrail
      R_Coil( "output"."2 层上行呼梯按钮指示灯" )
      R_Coil( "output"."1 号梯 1 层按钮指示灯" )
      R_Coil( "output"."1 号梯 1 级减速制动" )
      R_Coil( "output"."1 号梯 2 层按钮指示灯" )
      R_Coil( "output"."1 号梯 2 级减速制动" )
      R_Coil( "output"."1 号梯 3 层按钮指示灯" )
      R_Coil( "output"."1 号梯 3 级减速制动" )
      R_Coil( "output"."1 层上行呼梯按钮指示灯" )
   END_RUNG
   RUNG wire#powerrail
      R_Coil( "output"."1 号梯 5 层按钮指示灯" )
      R_Coil( "output"."1 号梯 6 层按钮指示灯" )
      R_Coil( "output"."1 号梯 LEDa" )
      R_Coil( "output"."1 号梯 LEDb" )
      R_Coil( "output"."1 号梯 LEDc" )
      R_Coil( "output"."1 号梯 LEDd" )
      R_Coil( "output"."1 号梯 LEDe" )
      R_Coil( "output"."1 号梯 4 层按钮指示灯" )
   END_RUNG
   RUNG wire#powerrail
      R_Coil( "output"."1 号梯 LEDg" )
      R_Coil( "output"."1 号梯 LEDf" )
      R_Coil( "output"."1 号梯低速接触器" )
      R_Coil( "output"."1 号梯风扇指示" )
      R_Coil( "output"."1 号梯高速接触器" )
      R_Coil( "output"."1 号梯故障指示" )
      R_Coil( "output"."1 号梯关门继电器" )
   END_RUNG
   RUNG wire#powerrail
      R_Coil( "output"."1 号梯满载指示" )
      "重置上下行"()
      R_Coil( "output"."1 号梯照明指示" )
      R_Coil( "output"."2 层下行呼梯按钮指示灯" )
      R_Coil( "output"."3 层上行呼梯按钮指示灯" )
      R_Coil( "output"."3 层下行呼梯按钮指示灯" )
      R_Coil( "output"."1 号梯开门继电器" )
   END_RUNG
   RUNG wire#powerrail
      R_Coil( "output"."4 层下行呼梯按钮指示灯" )
      R_Coil( "output"."5 层上行呼梯按钮指示灯" )
      R_Coil( "output"."5 层下行呼梯按钮指示灯" )
      R_Coil( "output"."6 层下行呼梯按钮指示灯" )
      R_Coil( "output"."4 层上行呼梯按钮指示灯" )
   END_RUNG
   // the same network as SCL:
   "output"."2 层上行呼梯按钮指示灯" := FALSE;
   "output"."1 号梯 1 层按钮指示灯" := FALSE;
   "output"."1 号梯 1 级减速制动" := FALSE;
   "output"."1 号梯 2 层按钮指示灯" := FALSE;
   "output"."1 号梯 2 级减速制动" := FALSE;
   "output"."1 号梯 3 层按钮指示灯" := FALSE;
   "output"."1 号梯 3 级减速制动" := FALSE;
   "output"."1 层上行呼梯按钮指示灯" := FALSE;
   "output"."1 号梯 5 层按钮指示灯" := FALSE;
   "output"."1 号梯 6 层按钮指示灯" := FALSE;
   "output"."1 号梯 LEDa" := FALSE;
   "output"."1 号梯 LEDb" := FALSE;
   "output"."1 号梯 LEDc" := FALSE;
   "output"."1 号梯 LEDd" := FALSE;
   "output"."1 号梯 LEDe" := FALSE;
   "output"."1 号梯 4 层按钮指示灯" := FALSE;
   "output"."1 号梯 LEDg" := FALSE;
   "output"."1 号梯 LEDf" := FALSE;
   "output"."1 号梯低速接触器" := FALSE;
   "output"."1 号梯风扇指示" := FALSE;
   "output"."1 号梯高速接触器" := FALSE;
   "output"."1 号梯故障指示" := FALSE;
   "output"."1 号梯关门继电器" := FALSE;
   "output"."1 号梯满载指示" := FALSE;
   "重置上下行"(ENO => #_w1);
   IF #_w1 THEN
       "output"."1 号梯照明指示" := FALSE;
       "output"."2 层下行呼梯按钮指示灯" := FALSE;
       "output"."3 层上行呼梯按钮指示灯" := FALSE;
       "output"."3 层下行呼梯按钮指示灯" := FALSE;
       "output"."1 号梯开门继电器" := FALSE;
   END_IF;
   "output"."4 层下行呼梯按钮指示灯" := FALSE;
   "output"."5 层上行呼梯按钮指示灯" := FALSE;
   "output"."5 层下行呼梯按钮指示灯" := FALSE;
   "output"."6 层下行呼梯按钮指示灯" := FALSE;
   "output"."4 层上行呼梯按钮指示灯" := FALSE;
END_REGION

REGION Network 2
   RUNG wire#powerrail
      Move(in := 0, out1 => "电梯上下行控制_DB_1".下行层数)
      Move(in := 0, out1 => "电梯上下行控制_DB_1".上升层数)
      Move(in := 0, out1 => "电梯上下行控制_DB_1".登记)
   END_RUNG
   // the same network as SCL:
   "电梯上下行控制_DB_1".下行层数 := 0;
   "电梯上下行控制_DB_1".上升层数 := 0;
   "电梯上下行控制_DB_1".登记 := 0;
END_REGION
END_FUNCTION

FUNCTION "楼层登记" : Void   // FC8, LAD
{ S7_Optimized_Access := 'TRUE' }
VERSION : 0.1
   VAR_INPUT
      楼层 : UInt;
      "上行/下行" : Bool;   // 上行为1，下行为0
   END_VAR
   VAR_TEMP
      tmp1 : Byte;
      tmp2 : Byte;
   END_VAR
   VAR_TEMP   // added for the SCL form of the ladder/FBD networks
      _w1 : Bool;
      _w2 : Bool;
      _w3 : Bool;
   END_VAR
BEGIN

REGION Network 1
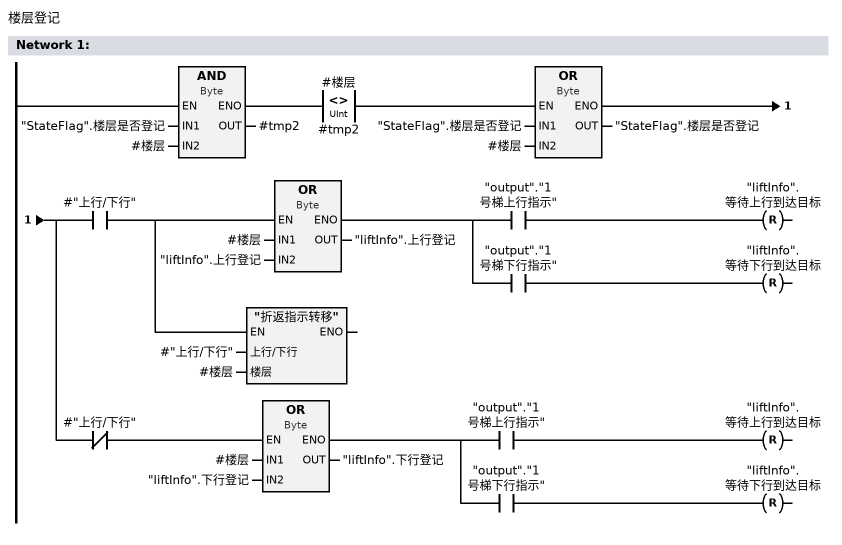
   #tmp2 := "StateFlag".楼层是否登记 AND #楼层;
   #_w1 := #楼层 <> #tmp2;
   IF #_w1 THEN "StateFlag".楼层是否登记 := "StateFlag".楼层是否登记 OR #楼层; END_IF;
   #_w2 := #_w1 AND #"上行/下行";
   IF #_w2 THEN "liftInfo".上行登记 := #楼层 OR "liftInfo".上行登记; END_IF;
   IF #_w2 AND "output"."1 号梯上行指示" THEN "liftInfo".等待上行到达目标 := FALSE; END_IF;
   IF #_w2 AND "output"."1 号梯下行指示" THEN "liftInfo".等待下行到达目标 := FALSE; END_IF;
   IF #_w2 THEN "折返指示转移"("上行/下行" := #"上行/下行", 楼层 := #楼层); END_IF;
   #_w3 := #_w1 AND NOT #"上行/下行";
   IF #_w3 THEN "liftInfo".下行登记 := #楼层 OR "liftInfo".下行登记; END_IF;
   IF #_w3 AND "output"."1 号梯上行指示" THEN "liftInfo".等待上行到达目标 := FALSE; END_IF;
   IF #_w3 AND "output"."1 号梯下行指示" THEN "liftInfo".等待下行到达目标 := FALSE; END_IF;
END_REGION
END_FUNCTION

FUNCTION "折返指示转移" : Void   // FC9, LAD
{ S7_Optimized_Access := 'TRUE' }
VERSION : 0.1
   VAR_INPUT
      "上行/下行" : Bool;
      楼层 : UInt;
   END_VAR
   VAR_TEMP
      tmp1 : Byte;
   END_VAR
   VAR_TEMP   // added for the SCL form of the ladder/FBD networks
      _w1 : Bool;
   END_VAR
BEGIN

REGION Network 1
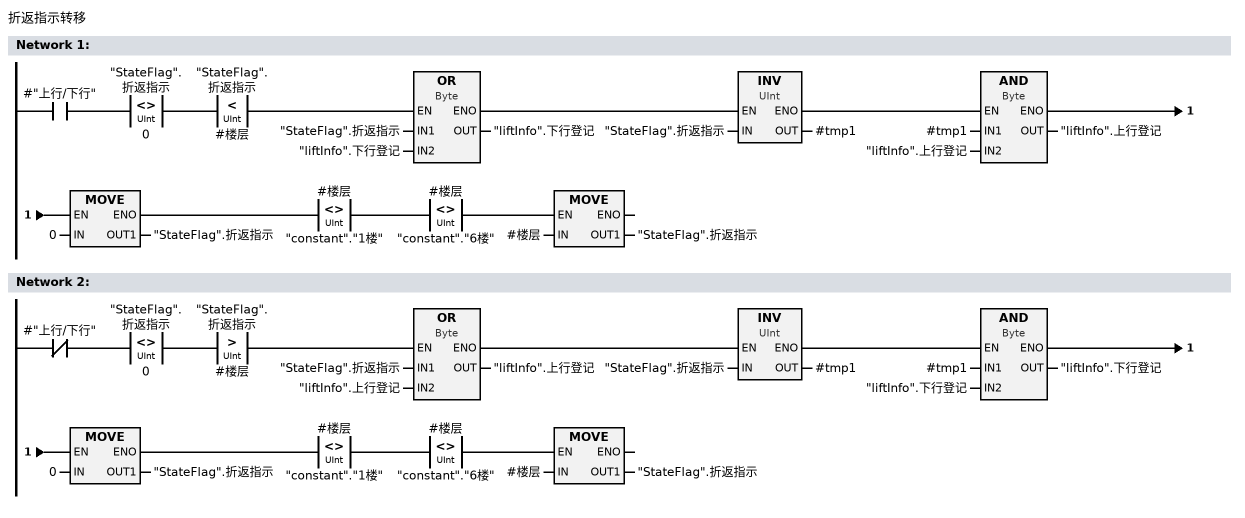
   #_w1 := #"上行/下行" AND ("StateFlag".折返指示 <> 0) AND ("StateFlag".折返指示 < #楼层);
   IF #_w1 THEN
       "liftInfo".下行登记 := "StateFlag".折返指示 OR "liftInfo".下行登记;
       #tmp1 := NOT "StateFlag".折返指示;
       "liftInfo".上行登记 := #tmp1 AND "liftInfo".上行登记;
       "StateFlag".折返指示 := 0;
   END_IF;
   IF #_w1 AND (#楼层 <> "constant"."1楼") AND (#楼层 <> "constant"."6楼") THEN "StateFlag".折返指示 := #楼层; END_IF;
END_REGION

REGION Network 2
   #_w1 := NOT #"上行/下行" AND ("StateFlag".折返指示 <> 0) AND ("StateFlag".折返指示 > #楼层);
   IF #_w1 THEN
       "liftInfo".上行登记 := "StateFlag".折返指示 OR "liftInfo".上行登记;
       #tmp1 := NOT "StateFlag".折返指示;
       "liftInfo".下行登记 := #tmp1 AND "liftInfo".下行登记;
       "StateFlag".折返指示 := 0;
   END_IF;
   IF #_w1 AND (#楼层 <> "constant"."1楼") AND (#楼层 <> "constant"."6楼") THEN "StateFlag".折返指示 := #楼层; END_IF;
END_REGION
END_FUNCTION

FUNCTION "循环左移" : Void   // FC10, LAD
{ S7_Optimized_Access := 'TRUE' }
VERSION : 0.1
// 循环左移1位
   VAR_INPUT
      掩码 : Byte;
   END_VAR
   VAR_IN_OUT
      数据 : Byte;
   END_VAR
   VAR_TEMP
      tmp1 : Byte;
   END_VAR
BEGIN

REGION Network 1
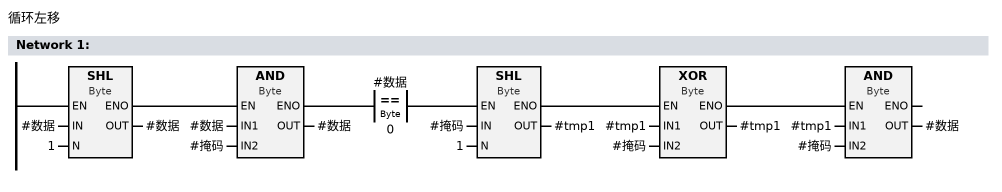
   #数据 := SHL(IN := #数据, N := 1);
   #数据 := #数据 AND #掩码;
   IF #数据 = 0 THEN
       #tmp1 := SHL(IN := #掩码, N := 1);
       #tmp1 := #tmp1 XOR #掩码;
       #数据 := #tmp1 AND #掩码;
   END_IF;
END_REGION
END_FUNCTION

FUNCTION "更新上下行掩码" : Void   // FC11, LAD
{ S7_Optimized_Access := 'TRUE' }
VERSION : 0.1
   VAR_TEMP
      tmp1 : Byte;
   END_VAR
BEGIN

REGION Network 1
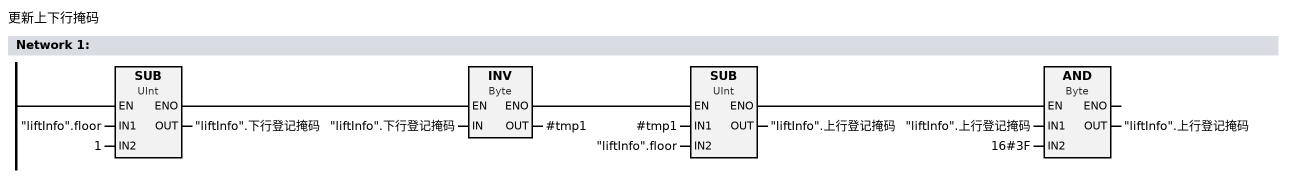
   RUNG wire#powerrail
      { S7_Templates := "SrcType := UInt" } Sub(in1 := "liftInfo".floor, in2 := 1, out => "liftInfo".下行登记掩码)
      { S7_Templates := "SrcType := Byte" } Inv(in := "liftInfo".下行登记掩码, out => #tmp1)
      { S7_Templates := "SrcType := UInt" } Sub(in1 := #tmp1, in2 := "liftInfo".floor, out => "liftInfo".上行登记掩码)
      { S7_Templates := "SrcType := Byte" } And(in1 := "liftInfo".上行登记掩码, in2 := 16#3F, out => "liftInfo".上行登记掩码)
   END_RUNG
   // the same network as SCL:
   "liftInfo".下行登记掩码 := "liftInfo".floor - 1;
   #tmp1 := NOT "liftInfo".下行登记掩码;
   "liftInfo".上行登记掩码 := #tmp1 - "liftInfo".floor;
   "liftInfo".上行登记掩码 := "liftInfo".上行登记掩码 AND 16#3F;
END_REGION
END_FUNCTION

ORGANIZATION_BLOCK "检修状态"   // OB1, LAD, ProgramCycle
TITLE = "Main Program Sweep (Cycle)"
{ S7_Optimized_Access := 'TRUE' }
VERSION : 0.1
   VAR_INPUT
      Initial_Call : Bool;   // Initial call of this OB
      Remanence : Bool;   // =True, if remanent data are available
   END_VAR
BEGIN

REGION Network 1
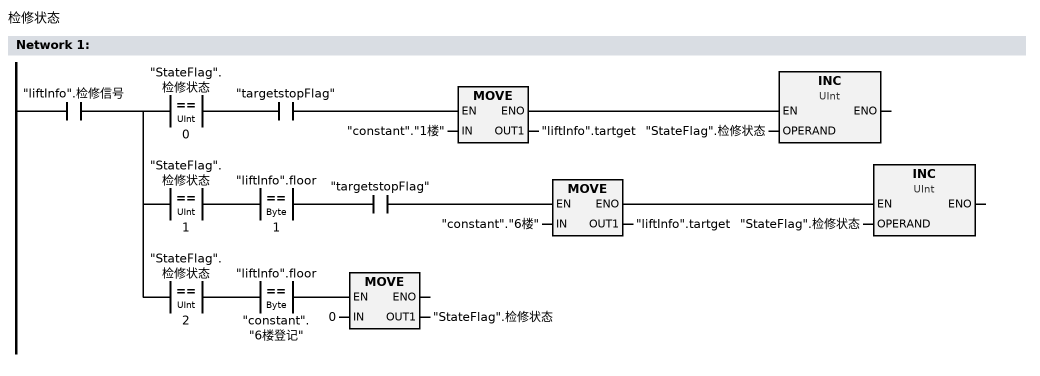
   RUNG wire#powerrail
      Contact( "liftInfo".检修信号 )
      wire#w1
      { S7_Templates := "SrcType := UInt" } EQ_Contact(in1 := "StateFlag".检修状态, in2 := 0)
      Contact( "targetstopFlag" )
      Move(in := "constant"."1楼", out1 => "liftInfo".tartget)
      { S7_Templates := "DestType := UInt" } Inc( "StateFlag".检修状态 )
   END_RUNG
   RUNG wire#w1
      { S7_Templates := "SrcType := UInt" } EQ_Contact(in1 := "StateFlag".检修状态, in2 := 1)
      { S7_Templates := "SrcType := Byte" } EQ_Contact(in1 := "liftInfo".floor, in2 := 1)
      Contact( "targetstopFlag" )
      Move(in := "constant"."6楼", out1 => "liftInfo".tartget)
      { S7_Templates := "DestType := UInt" } Inc( "StateFlag".检修状态 )
   END_RUNG
   RUNG wire#w1
      { S7_Templates := "SrcType := UInt" } EQ_Contact(in1 := "StateFlag".检修状态, in2 := 2)
      { S7_Templates := "SrcType := Byte" } EQ_Contact(in1 := "liftInfo".floor, in2 := "constant"."6楼登记")
      Move(in := 0, out1 => "StateFlag".检修状态)
   END_RUNG
   // the same network as SCL:
   IF "liftInfo".检修信号 AND ("StateFlag".检修状态 = 0) AND "targetstopFlag" THEN
       "liftInfo".tartget := "constant"."1楼";
       "StateFlag".检修状态 := "StateFlag".检修状态 + 1;
   END_IF;
   IF "liftInfo".检修信号 AND ("StateFlag".检修状态 = 1) AND ("liftInfo".floor = 1) AND "targetstopFlag" THEN
       "liftInfo".tartget := "constant"."6楼";
       "StateFlag".检修状态 := "StateFlag".检修状态 + 1;
   END_IF;
   IF "liftInfo".检修信号 AND ("StateFlag".检修状态 = 2) AND ("liftInfo".floor = "constant"."6楼登记") THEN
       "StateFlag".检修状态 := 0;
   END_IF;
END_REGION
END_ORGANIZATION_BLOCK

ORGANIZATION_BLOCK "Main"   // OB123, LAD, ProgramCycle
TITLE = "Main Program Sweep (Cycle)"
{ S7_Optimized_Access := 'TRUE' }
VERSION : 0.1
   VAR_INPUT
      Initial_Call : Bool;   // Initial call of this OB
      Remanence : Bool;   // =True, if remanent data are available
   END_VAR
   VAR_TEMP
      tmp1 : Byte;
      tmp2 : Byte;
      tmp3 : Byte;
   END_VAR
   VAR CONSTANT
      下行 : Bool;
      上行 : Bool := true;
   END_VAR
   VAR_TEMP   // added for the SCL form of the ladder/FBD networks
      _w1 : Bool;
      _w2 : Bool;
      _w3 : Bool;
      _w4 : Bool;
      _w5 : Bool;
      _w6 : Bool;
      _w7 : Bool;
      _w8 : Bool;
      _w9 : Bool;
   END_VAR
BEGIN

REGION Network 1: 指示灯
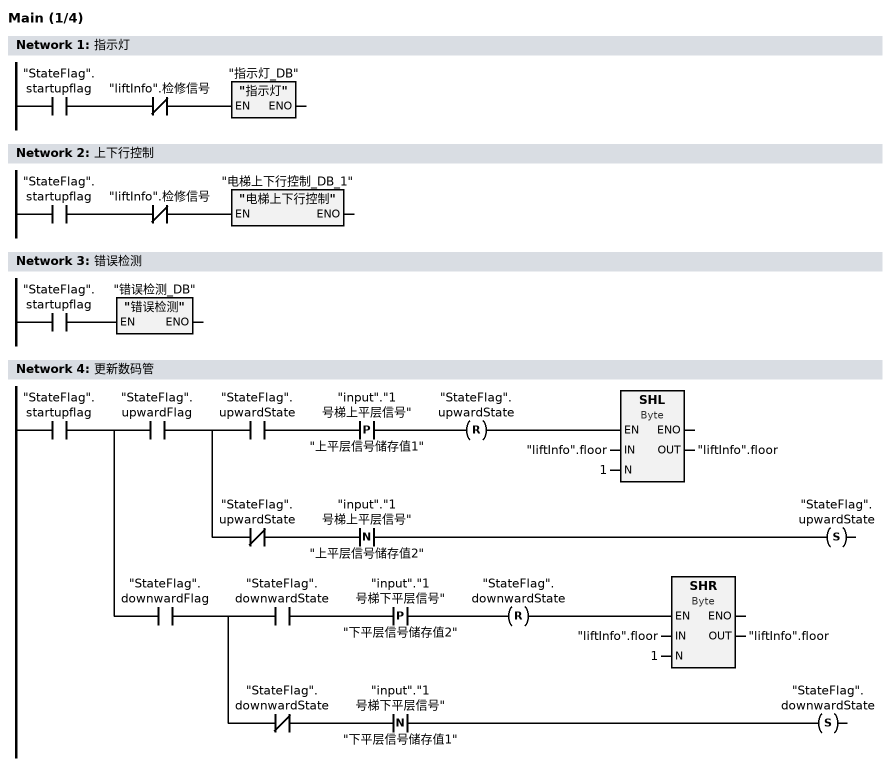
   RUNG wire#powerrail
      Contact( "StateFlag".startupflag )
      I_Contact( "liftInfo".检修信号 )
      "指示灯_DB"()
   END_RUNG
   // the same network as SCL:
   IF "StateFlag".startupflag AND NOT "liftInfo".检修信号 THEN
       "指示灯_DB"();   // "指示灯"
   END_IF;
END_REGION

REGION Network 2: 上下行控制
   RUNG wire#powerrail
      Contact( "StateFlag".startupflag )
      I_Contact( "liftInfo".检修信号 )
      "电梯上下行控制_DB_1"()
   END_RUNG
   // the same network as SCL:
   IF "StateFlag".startupflag AND NOT "liftInfo".检修信号 THEN
       "电梯上下行控制_DB_1"();   // "电梯上下行控制"
   END_IF;
END_REGION

REGION Network 3: 错误检测
   RUNG wire#powerrail
      Contact( "StateFlag".startupflag )
      "错误检测_DB"()
   END_RUNG
   // the same network as SCL:
   IF "StateFlag".startupflag THEN
       "错误检测_DB"();   // "错误检测"
   END_IF;
END_REGION

REGION Network 4: 更新数码管
   RUNG wire#powerrail
      Contact( "StateFlag".startupflag )
      wire#w1
      Contact( "StateFlag".upwardFlag )
      wire#w2
      Contact( "StateFlag".upwardState )
      P_Contact(operand := "input"."1 号梯上平层信号", bit := "上平层信号储存值1")
      R_Coil( "StateFlag".upwardState )
      { S7_Templates := "SrcType := Byte" } Shl(in := "liftInfo".floor, n := 1, out => "liftInfo".floor)
   END_RUNG
   RUNG wire#w2
      I_Contact( "StateFlag".upwardState )
      N_Contact(operand := "input"."1 号梯上平层信号", bit := "上平层信号储存值2")
      S_Coil( "StateFlag".upwardState )
   END_RUNG
   RUNG wire#w1
      Contact( "StateFlag".downwardFlag )
      wire#w3
      Contact( "StateFlag".downwardState )
      P_Contact(operand := "input"."1 号梯下平层信号", bit := "下平层信号储存值2")
      R_Coil( "StateFlag".downwardState )
      { S7_Templates := "SrcType := Byte" } Shr(in := "liftInfo".floor, n := 1, out => "liftInfo".floor)
   END_RUNG
   RUNG wire#w3
      I_Contact( "StateFlag".downwardState )
      N_Contact(operand := "input"."1 号梯下平层信号", bit := "下平层信号储存值1")
      S_Coil( "StateFlag".downwardState )
   END_RUNG
   // the same network as SCL:
   #_w1 := "StateFlag".startupflag AND "StateFlag".upwardFlag;
   #_w2 := #_w1 AND "StateFlag".upwardState AND "input"."1 号梯上平层信号" AND NOT "上平层信号储存值1";   // rising edge of "input"."1 号梯上平层信号"
   "上平层信号储存值1" := "input"."1 号梯上平层信号";
   IF #_w2 THEN
       "StateFlag".upwardState := FALSE;
       "liftInfo".floor := SHL(IN := "liftInfo".floor, N := 1);
   END_IF;
   #_w3 := #_w1 AND NOT "StateFlag".upwardState AND NOT "input"."1 号梯上平层信号" AND "上平层信号储存值2";   // falling edge of "input"."1 号梯上平层信号"
   "上平层信号储存值2" := "input"."1 号梯上平层信号";
   IF #_w3 THEN "StateFlag".upwardState := TRUE; END_IF;
   #_w4 := "StateFlag".startupflag AND "StateFlag".downwardFlag;
   #_w5 := #_w4 AND "StateFlag".downwardState AND "input"."1 号梯下平层信号" AND NOT "下平层信号储存值2";   // rising edge of "input"."1 号梯下平层信号"
   "下平层信号储存值2" := "input"."1 号梯下平层信号";
   IF #_w5 THEN
       "StateFlag".downwardState := FALSE;
       "liftInfo".floor := SHR(IN := "liftInfo".floor, N := 1);
   END_IF;
   #_w6 := #_w4 AND NOT "StateFlag".downwardState AND NOT "input"."1 号梯下平层信号" AND "下平层信号储存值1";   // falling edge of "input"."1 号梯下平层信号"
   "下平层信号储存值1" := "input"."1 号梯下平层信号";
   IF #_w6 THEN "StateFlag".downwardState := TRUE; END_IF;
END_REGION

REGION Network 5: 前往指定楼层
